KUKA KRL program: MyProgram_158().src

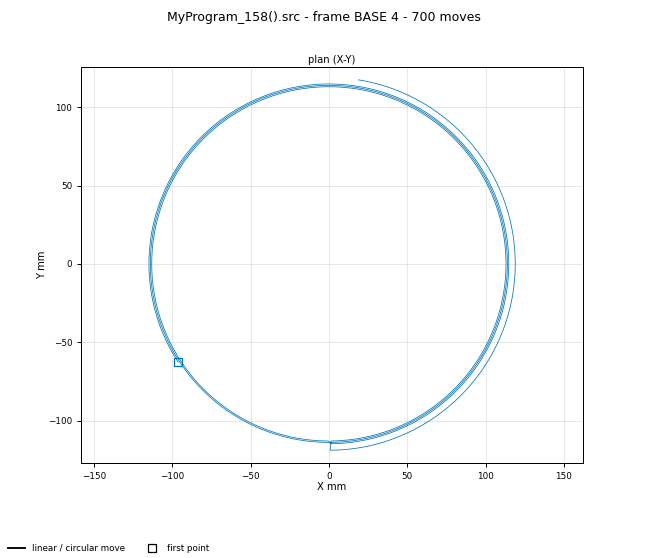
[picture p0: tool path of MyProgram_158().src in frame BASE 4, 700 of 700 moves have a stored position in this frame; points joined in program order, loops and branches not executed]
&ACCESS RVP
&REL 1
&PARAM TEMPLATE = C:\KRC\Roboter\Template\vorgabe
&PARAM EDITMASK = *
DEF MyProgram_158()
; ---- Setting reference (Base) ----
$BASE = BASE_DATA[4]

; --------------------------
; ---- Setting tool (TCP) ----
$TOOL = TOOL_DATA[3]
; --------------------------

$VEL.CP = VEL_APROX_PRINT
Startdeposition()
$VEL.CP = VEL_PRINT
LIN {X -96.1215,Y -62.8058,Z 121,A -151.3132,B 24.9534,C -1.5764,E1 24.8649,E2 237.3764} C_DIS
LIN {X -98.7062,Y -58.6591,Z 121,A -153.4833,B 24.9524,C -1.5937,E1 24.8618,E2 239.5163} C_DIS
LIN {X -100.613,Y -55.328,Z 121,A -155.5079,B 24.9524,C -1.5945,E1 24.859,E2 241.5496} C_DIS
LIN {X -102.3262,Y -52.0874,Z 121,A -157.2957,B 24.952,C -1.6013,E1 24.8567,E2 243.3308} C_DIS
LIN {X -104.3543,Y -47.8986,Z 121,A -160.2123,B 24.953,C -1.5842,E1 24.8532,E2 246.3041} C_DIS
LIN {X -106.1362,Y -43.808,Z 121,A -161.886,B 24.9513,C -1.6127,E1 24.8515,E2 247.9191} C_DIS
LIN {X -107.2271,Y -41.0641,Z 121,A -163.2123,B 24.9506,C -1.6229,E1 24.8501,E2 249.2284} C_DIS
LIN {X -108.5471,Y -37.4383,Z 121,A -165.2668,B 24.9506,C -1.6235,E1 24.8482,E2 251.2933} C_DIS
LIN {X -109.6661,Y -34.0158,Z 121,A -167.0294,B 24.9502,C -1.6304,E1 24.8467,E2 253.0496} C_DIS
LIN {X -110.6984,Y -30.4946,Z 121,A -168.9363,B 24.95,C -1.6329,E1 24.8452,E2 254.9614} C_DIS
LIN {X -111.5787,Y -27.0914,Z 121,A -170.6546,B 24.9496,C -1.6398,E1 24.8441,E2 256.6733} C_DIS
LIN {X -112.4202,Y -23.3559,Z 121,A -172.6551,B 24.9495,C -1.6422,E1 24.8429,E2 258.6799} C_DIS
LIN {X -113.0351,Y -20.1694,Z 121,A -174.8026,B 24.9504,C -1.6265,E1 24.8418,E2 260.8777} C_DIS
LIN {X -113.7096,Y -15.9343,Z 121,A -176.449,B 24.9488,C -1.6528,E1 24.8412,E2 262.4712} C_DIS
LIN {X -114.0425,Y -13.3431,Z 121,A -178.2058,B 24.9497,C -1.6391,E1 24.8406,E2 264.2712} C_DIS
LIN {X -114.4392,Y -9.3513,Z 121,A 179.6628,B 24.9496,C -1.6404,E1 24.8401,E2 266.4122} C_DIS
LIN {X -114.7175,Y -4.8606,Z 121,A 178.0279,B 24.9476,C -1.6717,E1 24.8399,E2 267.9823} C_DIS
LIN {X -114.814,Y -1.3829,Z 121,A 175.4927,B 24.9492,C -1.6459,E1 24.8399,E2 270.5943} C_DIS
LIN {X -114.7594,Y 3.7508,Z 121,A 173.0506,B 24.9484,C -1.659,E1 24.84,E2 273.02} C_DIS
LIN {X -114.514,Y 8.3994,Z 121,A 171.3096,B 24.9465,C -1.6894,E1 24.8403,E2 274.699} C_DIS
LIN {X -113.8679,Y 14.7586,Z 121,A 168.0814,B 24.946,C -1.6982,E1 24.8413,E2 277.9254} C_DIS
LIN {X -113.3453,Y 18.3552,Z 121,A 166.2551,B 24.9456,C -1.7036,E1 24.8421,E2 279.7497} C_DIS
LIN {X -112.7131,Y 21.898,Z 121,A 164.4701,B 24.9452,C -1.7098,E1 24.843,E2 281.5304} C_DIS
LIN {X -112.1059,Y 24.8216,Z 121,A 162.4049,B 24.9463,C -1.692,E1 24.8443,E2 283.6503} C_DIS
LIN {X -111.0532,Y 29.1768,Z 121,A 160.7315,B 24.9445,C -1.7213,E1 24.8454,E2 285.2636} C_DIS
LIN {X -110.14,Y 32.4493,Z 121,A 159.1356,B 24.9439,C -1.7306,E1 24.8466,E2 286.8465} C_DIS
LIN {X -107.4375,Y 40.5085,Z 121,A 154.9999,B 24.9427,C -1.7481,E1 24.8503,E2 290.964} C_DIS
LIN {X -105.096,Y 46.2461,Z 121,A 151.596,B 24.9429,C -1.7452,E1 24.854,E2 294.3938} C_DIS
LIN {X -102.9973,Y 50.7479,Z 121,A 149.1343,B 24.9424,C -1.7534,E1 24.8569,E2 296.8493} C_DIS
LIN {X -101.2249,Y 54.1999,Z 121,A 147.1466,B 24.9421,C -1.7571,E1 24.8595,E2 298.8389} C_DIS
LIN {X -96.7746,Y 61.7938,Z 121,A 142.7854,B 24.9412,C -1.771,E1 24.8658,E2 303.1894} C_DIS
LIN {X -94.9438,Y 64.5713,Z 121,A 140.5435,B 24.9424,C -1.7526,E1 24.8694,E2 305.4863} C_DIS
LIN {X -92.4138,Y 68.1437,Z 121,A 138.3387,B 24.9421,C -1.7578,E1 24.873,E2 307.6894} C_DIS
LIN {X -89.7147,Y 71.6613,Z 121,A 136.6412,B 24.9403,C -1.7841,E1 24.8758,E2 309.3321} C_DIS
LIN {X -87.3156,Y 74.5636,Z 121,A 134.8321,B 24.9398,C -1.7919,E1 24.8791,E2 311.1311} C_DIS
LIN {X -84.7529,Y 77.4644,Z 121,A 132.9066,B 24.9395,C -1.797,E1 24.8826,E2 313.0529} C_DIS
LIN {X -82.5435,Y 79.8143,Z 121,A 131.2955,B 24.9392,C -1.801,E1 24.8857,E2 314.6615} C_DIS
LIN {X -79.9211,Y 82.4406,Z 121,A 129.4166,B 24.939,C -1.8044,E1 24.8895,E2 316.5402} C_DIS
LIN {X -77.5694,Y 84.6565,Z 121,A 127.7878,B 24.9388,C -1.8075,E1 24.8928,E2 318.1682} C_DIS
LIN {X -74.6448,Y 87.2464,Z 121,A 125.8351,B 24.9385,C -1.8119,E1 24.8969,E2 320.1183} C_DIS
LIN {X -72.0721,Y 89.3835,Z 121,A 124.0608,B 24.9385,C -1.8113,E1 24.9008,E2 321.9006} C_DIS
LIN {X -68.9305,Y 91.8277,Z 121,A 122.1405,B 24.938,C -1.8182,E1 24.905,E2 323.8114} C_DIS
LIN {X -64.5217,Y 94.9774,Z 121,A 119.0522,B 24.9387,C -1.8081,E1 24.9122,E2 326.9343} C_DIS
LIN {X -61.6039,Y 96.8965,Z 121,A 117.6079,B 24.9377,C -1.8235,E1 24.9155,E2 328.3465} C_DIS
LIN {X -58.7884,Y 98.6297,Z 121,A 115.9289,B 24.9375,C -1.8254,E1 24.9195,E2 330.0263} C_DIS
LIN {X -55.2102,Y 100.6769,Z 121,A 114.0202,B 24.9369,C -1.8351,E1 24.9241,E2 331.9175} C_DIS
LIN {X -52.7307,Y 101.9975,Z 121,A 112.5738,B 24.9369,C -1.8356,E1 24.9277,E2 333.3666} C_DIS
LIN {X -50.4381,Y 103.1509,Z 121,A 110.373,B 24.9393,C -1.8001,E1 24.9335,E2 335.6574} C_DIS
LIN {X -45.2421,Y 105.5337,Z 121,A 108.4902,B 24.9363,C -1.844,E1 24.938,E2 337.4405} C_DIS
LIN {X -39.388,Y 107.8532,Z 121,A 105.2389,B 24.9363,C -1.8437,E1 24.9465,E2 340.6993} C_DIS
LIN {X -35.8676,Y 109.0758,Z 121,A 103.4013,B 24.9361,C -1.8469,E1 24.9513,E2 342.5329} C_DIS
LIN {X -32.6704,Y 110.0744,Z 121,A 101.7237,B 24.9359,C -1.8486,E1 24.9558,E2 344.2094} C_DIS
LIN {X -28.9554,Y 111.1101,Z 121,A 99.5825,B 24.9364,C -1.8415,E1 24.9616,E2 346.3706} C_DIS
LIN {X -23.8184,Y 112.3248,Z 121,A 96.5727,B 24.9373,C -1.8283,E1 24.9699,E2 349.4157} C_DIS
LIN {X -19.6037,Y 113.1365,Z 121,A 94.9134,B 24.9358,C -1.85,E1 24.9744,E2 351.025} C_DIS
LIN {X -13.3544,Y 114.0412,Z 121,A 92.0278,B 24.9349,C -1.8632,E1 24.9823,E2 353.8815} C_DIS
LIN {X -7.8614,Y 114.551,Z 121,A 89.1574,B 24.9352,C -1.8595,E1 24.9903,E2 356.762} C_DIS
LIN {X -4.8853,Y 114.7164,Z 121,A 86.9827,B 24.9372,C -1.831,E1 24.9966,E2 359.0049} C_DIS
LIN {X -0.3746,Y 114.8203,Z 121,A 85.6519,B 24.9344,C -1.8706,E1 25,E2 360.242} C_DIS
LIN {X 5.1557,Y 114.7048,Z 121,A 82.5408,B 24.9354,C -1.8558,E1 25.0088,E2 363.3874} C_DIS
LIN {X 7.8335,Y 114.5529,Z 121,A 80.6882,B 24.937,C -1.8339,E1 25.0141,E2 365.2913} C_DIS
LIN {X 12.0548,Y 114.1859,Z 121,A 78.4447,B 24.9374,C -1.8281,E1 25.0203,E2 367.5469} C_DIS
LIN {X 16.9074,Y 113.5706,Z 121,A 76.5126,B 24.9359,C -1.8491,E1 25.0255,E2 369.4275} C_DIS
LIN {X 21.8894,Y 112.7147,Z 121,A 74.2506,B 24.9352,C -1.8594,E1 25.0317,E2 371.6625} C_DIS
LIN {X 26.0769,Y 111.8203,Z 121,A 72.0876,B 24.9353,C -1.8572,E1 25.0376,E2 373.8279} C_DIS
LIN {X 29.1301,Y 111.0652,Z 121,A 70.5499,B 24.9353,C -1.8576,E1 25.0417,E2 375.3623} C_DIS
LIN {X 33.9752,Y 109.6787,Z 121,A 67.9832,B 24.9356,C -1.8535,E1 25.0486,E2 377.9344} C_DIS
LIN {X 37.6505,Y 108.4726,Z 121,A 65.9823,B 24.9359,C -1.8488,E1 25.0539,E2 379.9426} C_DIS
LIN {X 41.1905,Y 107.1792,Z 121,A 64.0737,B 24.9361,C -1.8457,E1 25.0589,E2 381.8543} C_DIS
LIN {X 44.6995,Y 105.7625,Z 121,A 62.3212,B 24.9359,C -1.8497,E1 25.0634,E2 383.5933} C_DIS
LIN {X 48.0774,Y 104.2711,Z 121,A 60.4926,B 24.9359,C -1.8482,E1 25.0681,E2 385.421} C_DIS
LIN {X 51.8809,Y 102.4318,Z 121,A 58.3052,B 24.9364,C -1.842,E1 25.0736,E2 387.6171} C_DIS
LIN {X 55.0868,Y 100.7438,Z 121,A 56.5389,B 24.9364,C -1.8414,E1 25.0779,E2 389.3798} C_DIS
LIN {X 58.2725,Y 98.9347,Z 121,A 54.7042,B 24.9366,C -1.8385,E1 25.0824,E2 391.2159} C_DIS
LIN {X 61.4356,Y 97.0046,Z 121,A 52.8073,B 24.937,C -1.8335,E1 25.0869,E2 393.1187} C_DIS
LIN {X 63.9947,Y 95.3342,Z 121,A 51.3249,B 24.937,C -1.8329,E1 25.0903,E2 394.5976} C_DIS
LIN {X 66.3478,Y 93.7116,Z 121,A 49.8719,B 24.9373,C -1.8293,E1 25.0936,E2 396.0541} C_DIS
LIN {X 69.4672,Y 91.4244,Z 121,A 46.9689,B 24.9404,C -1.7825,E1 25.1003,E2 399.0569} C_DIS
LIN {X 74.3586,Y 87.4903,Z 121,A 45.2175,B 24.9367,C -1.8382,E1 25.1038,E2 400.6701} C_DIS
LIN {X 78.1942,Y 84.0821,Z 121,A 42.2735,B 24.9382,C -1.8156,E1 25.11,E2 403.6558} C_DIS
LIN {X 80.7429,Y 81.6353,Z 121,A 40.602,B 24.9382,C -1.816,E1 25.1133,E2 405.3193} C_DIS
LIN {X 82.4406,Y 79.9211,Z 121,A 38.63,B 24.9407,C -1.7787,E1 25.1173,E2 407.3707} C_DIS
LIN {X 85.9184,Y 76.1709,Z 121,A 36.8868,B 24.9386,C -1.8094,E1 25.1204,E2 409.0339} C_DIS
LIN {X 89.5047,Y 71.9227,Z 121,A 33.9906,B 24.9395,C -1.7972,E1 25.1256,E2 411.9455} C_DIS
LIN {X 91.5655,Y 69.2794,Z 121,A 32.4088,B 24.9395,C -1.7972,E1 25.1283,E2 413.5196} C_DIS
LIN {X 93.5687,Y 66.5482,Z 121,A 30.7815,B 24.9395,C -1.7959,E1 25.1309,E2 415.1423} C_DIS
LIN {X 96.4611,Y 62.2823,Z 121,A 28.1901,B 24.9401,C -1.7883,E1 25.135,E2 417.7387} C_DIS
LIN {X 98.3019,Y 59.3344,Z 121,A 26.397,B 24.9405,C -1.781,E1 25.1376,E2 419.54} C_DIS
LIN {X 99.997,Y 56.4322,Z 121,A 24.8055,B 24.9405,C -1.7803,E1 25.1398,E2 421.1248} C_DIS
LIN {X 101.6157,Y 53.46,Z 121,A 22.5104,B 24.9427,C -1.7479,E1 25.1429,E2 423.4843} C_DIS
LIN {X 103.598,Y 49.51,Z 121,A 20.5831,B 24.9423,C -1.7543,E1 25.1452,E2 425.3861} C_DIS
LIN {X 104.9951,Y 46.4775,Z 121,A 19.1792,B 24.9418,C -1.7615,E1 25.1467,E2 426.7654} C_DIS
LIN {X 106.3722,Y 43.2284,Z 121,A 17.5035,B 24.9419,C -1.7603,E1 25.1485,E2 428.4347} C_DIS
LIN {X 107.8329,Y 39.4436,Z 121,A 15.5282,B 24.9422,C -1.7566,E1 25.1505,E2 430.4078} C_DIS
LIN {X 109.0136,Y 36.0582,Z 121,A 13.8068,B 24.9423,C -1.7543,E1 25.152,E2 432.1249} C_DIS
LIN {X 110.5926,Y 30.8741,Z 121,A 10.9602,B 24.9433,C -1.7394,E1 25.1543,E2 434.9904} C_DIS
LIN {X 111.6671,Y 26.7289,Z 121,A 8.5014,B 24.9447,C -1.7178,E1 25.156,E2 437.4858} C_DIS
LIN {X 112.4325,Y 23.296,Z 121,A 7.1876,B 24.9437,C -1.7328,E1 25.1567,E2 438.7567} C_DIS
LIN {X 112.9625,Y 20.5735,Z 121,A 5.3858,B 24.9453,C -1.709,E1 25.1576,E2 440.604} C_DIS
LIN {X 113.558,Y 16.9887,Z 121,A 3.9219,B 24.9446,C -1.7194,E1 25.1582,E2 442.0348} C_DIS
LIN {X 114.0229,Y 13.5104,Z 121,A 2.2875,B 24.9446,C -1.7193,E1 25.1588,E2 443.66} C_DIS
LIN {X 114.3753,Y 10.1102,Z 121,A 0.5482,B 24.9451,C -1.7122,E1 25.1593,E2 445.4056} C_DIS
LIN {X 114.6333,Y 6.5551,Z 121,A -1.1978,B 24.9453,C -1.708,E1 25.1596,E2 447.1512} C_DIS
LIN {X 114.7743,Y 3.2623,Z 121,A -2.8664,B 24.9457,C -1.7015,E1 25.1598,E2 448.8251} C_DIS
LIN {X 114.8185,Y -0.7449,Z 121,A -4.8494,B 24.9461,C -1.6957,E1 25.1598,E2 450.8098} C_DIS
LIN {X 114.7256,Y -4.6719,Z 121,A -6.7449,B 24.9463,C -1.6924,E1 25.1596,E2 452.702} C_DIS
LIN {X 114.5495,Y -7.8841,Z 121,A -8.3454,B 24.9466,C -1.6874,E1 25.1593,E2 454.3049} C_DIS
LIN {X 114.2214,Y -11.7158,Z 121,A -9.9878,B 24.9462,C -1.6941,E1 25.1589,E2 455.9217} C_DIS
LIN {X 113.6208,Y -16.5537,Z 121,A -13.0095,B 24.9485,C -1.6586,E1 25.1578,E2 459.0092} C_DIS
LIN {X 113.104,Y -19.7867,Z 121,A -14.3439,B 24.9479,C -1.6672,E1 25.1572,E2 460.3155} C_DIS
LIN {X 112.5322,Y -22.8105,Z 121,A -15.8061,B 24.948,C -1.6657,E1 25.1564,E2 461.7727} C_DIS
LIN {X 112.0044,Y -25.28,Z 121,A -17.0567,B 24.9482,C -1.662,E1 25.1556,E2 463.0247} C_DIS
LIN {X 111.2159,Y -28.5439,Z 121,A -18.737,B 24.9486,C -1.6564,E1 25.1545,E2 464.7084} C_DIS
LIN {X 110.2966,Y -31.9185,Z 121,A -20.5716,B 24.9492,C -1.6466,E1 25.1531,E2 466.5557} C_DIS
LIN {X 109.2307,Y -35.3889,Z 121,A -22.6194,B 24.9502,C -1.6299,E1 25.1514,E2 468.6313} C_DIS
LIN {X 108.1578,Y -38.5478,Z 121,A -24.0023,B 24.9497,C -1.6378,E1 25.1501,E2 469.9878} C_DIS
LIN {X 106.8943,Y -41.9206,Z 121,A -25.5185,B 24.9493,C -1.6453,E1 25.1486,E2 471.4778} C_DIS
LIN {X 105.7281,Y -44.781,Z 121,A -27.3593,B 24.9504,C -1.6265,E1 25.1466,E2 473.3527} C_DIS
LIN {X 102.7462,Y -51.2545,Z 121,A -30.8679,B 24.9509,C -1.6179,E1 25.1424,E2 476.8627} C_DIS
LIN {X 100.9603,Y -54.6877,Z 121,A -32.4978,B 24.9504,C -1.6262,E1 25.1403,E2 478.4645} C_DIS
LIN {X 97.0688,Y -61.3329,Z 121,A -36.5884,B 24.9518,C -1.6034,E1 25.1345,E2 482.5879} C_DIS
LIN {X 95.0203,Y -64.4584,Z 121,A -38.3723,B 24.9519,C -1.6019,E1 25.1317,E2 484.3666} C_DIS
LIN {X 92.7868,Y -67.6343,Z 121,A -40.2813,B 24.9522,C -1.5978,E1 25.1286,E2 486.2759} C_DIS
LIN {X 90.7135,Y -70.3913,Z 121,A -42.0985,B 24.9527,C -1.5886,E1 25.1255,E2 488.1061} C_DIS
LIN {X 88.3561,Y -73.3275,Z 121,A -43.8607,B 24.9527,C -1.589,E1 25.1224,E2 489.8592} C_DIS
LIN {X 86.0399,Y -76.0345,Z 121,A -45.7192,B 24.9532,C -1.5806,E1 25.119,E2 491.7291} C_DIS
LIN {X 83.5677,Y -78.7413,Z 121,A -47.4804,B 24.9532,C -1.5791,E1 25.1156,E2 493.4862} C_DIS
LIN {X 80.6526,Y -81.7245,Z 121,A -49.7015,B 24.954,C -1.5676,E1 25.1112,E2 495.7251} C_DIS
LIN {X 77.4731,Y -84.7448,Z 121,A -51.6968,B 24.9537,C -1.5712,E1 25.1072,E2 497.7036} C_DIS
LIN {X 74.7706,Y -87.1392,Z 121,A -53.5625,B 24.9542,C -1.5641,E1 25.1033,E2 499.5788} C_DIS
LIN {X 69.9227,Y -91.0746,Z 121,A -56.6293,B 24.9544,C -1.5594,E1 25.0966,E2 502.6451} C_DIS
LIN {X 66.8672,Y -93.341,Z 121,A -58.4819,B 24.9545,C -1.5575,E1 25.0924,E2 504.4957} C_DIS
LIN {X 64.0295,Y -95.3107,Z 121,A -60.3186,B 24.9551,C -1.5489,E1 25.0881,E2 506.3466} C_DIS
LIN {X 60.7768,Y -97.4161,Z 121,A -62.1258,B 24.9549,C -1.5509,E1 25.0839,E2 508.1433} C_DIS
LIN {X 57.5124,Y -99.379,Z 121,A -63.84,B 24.9546,C -1.5558,E1 25.0798,E2 509.8404} C_DIS
LIN {X 54.723,Y -100.9412,Z 121,A -66.578,B 24.9578,C -1.5015,E1 25.0728,E2 512.6989} C_DIS
LIN {X 49.393,Y -103.6542,Z 121,A -68.4656,B 24.9552,C -1.5458,E1 25.0683,E2 514.4767} C_DIS
LIN {X 42.3067,Y -106.7426,Z 121,A -72.4489,B 24.9559,C -1.5343,E1 25.0581,E2 518.4777} C_DIS
LIN {X 39.0113,Y -107.9906,Z 121,A -74.2842,B 24.9562,C -1.5285,E1 25.0532,E2 520.323} C_DIS
LIN {X 35.716,Y -109.1249,Z 121,A -75.866,B 24.956,C -1.5333,E1 25.0491,E2 521.8902} C_DIS
LIN {X 30.3415,Y -110.7397,Z 121,A -78.6548,B 24.9561,C -1.5307,E1 25.0416,E2 524.6806} C_DIS
LIN {X 27.6754,Y -111.4362,Z 121,A -80.0133,B 24.9561,C -1.53,E1 25.0379,E2 526.0386} C_DIS
LIN {X 21.6881,Y -112.7535,Z 121,A -83.0024,B 24.9561,C -1.5303,E1 25.0298,E2 529.023} C_DIS
LIN {X 15.8742,Y -113.7181,Z 121,A -86.1649,B 24.9568,C -1.5183,E1 25.021,E2 532.211} C_DIS
LIN {X 11.583,Y -114.2353,Z 121,A -88.3362,B 24.9569,C -1.5163,E1 25.015,E2 534.3853} C_DIS
LIN {X 7.9927,Y -114.5422,Z 121,A -89.9911,B 24.9566,C -1.5218,E1 25.0104,E2 536.0265} C_DIS
LIN {X 5.0588,Y -114.709,Z 121,A -91.4832,B 24.9567,C -1.5201,E1 25.0062,E2 537.5222} C_DIS
LIN {X 1.4985,Y -114.8123,Z 121,A -93.3515,B 24.957,C -1.5155,E1 25.001,E2 539.4009} C_DIS
LIN {X 1.4985,Y -114.8123,Z 121,A -93.3515,B 24.957,C -1.5155,E1 25.001,E2 539.4009} C_DIS
Enddeposition()
LIN {X 0.8205,Y -113.9352,Z 121,A -93.6003,B 24.9559,C -1.5349,E1 25.0004,E2 539.6037} C_DIS
Startdeposition()
$VEL.CP = VEL_PRINT
LIN {X 4.8717,Y -113.8345,Z 121,A -90.8478,B 24.954,C -1.5668,E1 25.0083,E2 536.7761} C_DIS
LIN {X 8.1536,Y -113.6476,Z 121,A -89.0673,B 24.9536,C -1.5732,E1 25.0133,E2 534.9813} C_DIS
LIN {X 14.6994,Y -112.9866,Z 121,A -86.2906,B 24.9549,C -1.5515,E1 25.0209,E2 532.2578} C_DIS
LIN {X 20.9577,Y -111.9963,Z 121,A -82.4435,B 24.953,C -1.5833,E1 25.0317,E2 528.3394} C_DIS
LIN {X 26.0634,Y -110.9185,Z 121,A -80.1548,B 24.9538,C -1.5707,E1 25.0378,E2 526.0835} C_DIS
LIN {X 29.0685,Y -110.1703,Z 121,A -78.6045,B 24.9538,C -1.572,E1 25.042,E2 524.5326} C_DIS
LIN {X 32.1861,Y -109.2984,Z 121,A -76.7232,B 24.9529,C -1.5852,E1 25.0471,E2 522.6231} C_DIS
LIN {X 36.1944,Y -108.0373,Z 121,A -74.8013,B 24.9533,C -1.5792,E1 25.0522,E2 520.719} C_DIS
LIN {X 39.2027,Y -106.9823,Z 121,A -73.2543,B 24.9533,C -1.5788,E1 25.0562,E2 519.1763} C_DIS
LIN {X 42.4649,Y -105.731,Z 121,A -70.9958,B 24.9518,C -1.604,E1 25.0623,E2 516.863} C_DIS
LIN {X 45.7854,Y -104.3351,Z 121,A -69.8746,B 24.9535,C -1.5754,E1 25.065,E2 515.8122} C_DIS
LIN {X 47.9547,Y -103.3557,Z 121,A -68.446,B 24.9528,C -1.5878,E1 25.0686,E2 514.358} C_DIS
LIN {X 51.2356,Y -101.7713,Z 121,A -66.5435,B 24.9524,C -1.594,E1 25.0734,E2 512.4459} C_DIS
LIN {X 56.7317,Y -98.8107,Z 121,A -63.5306,B 24.9524,C -1.5938,E1 25.0808,E2 509.4423} C_DIS
LIN {X 59.3692,Y -97.2491,Z 121,A -61.9362,B 24.9521,C -1.5991,E1 25.0846,E2 507.8403} C_DIS
LIN {X 62.7529,Y -95.1005,Z 121,A -59.9229,B 24.9519,C -1.6029,E1 25.0893,E2 505.8244} C_DIS
LIN {X 65.6081,Y -93.1563,Z 121,A -58.2849,B 24.9519,C -1.6019,E1 25.0931,E2 504.1945} C_DIS
LIN {X 67.4533,Y -91.8265,Z 121,A -57.1559,B 24.9519,C -1.6037,E1 25.0956,E2 503.0654} C_DIS
LIN {X 70.0049,Y -89.8982,Z 121,A -55.2667,B 24.9508,C -1.6201,E1 25.0999,E2 501.1442} C_DIS
LIN {X 72.7486,Y -87.6908,Z 121,A -53.7199,B 24.9512,C -1.6137,E1 25.1032,E2 499.6184} C_DIS
LIN {X 75.2244,Y -85.5772,Z 121,A -52.1275,B 24.9512,C -1.6154,E1 25.1065,E2 498.0282} C_DIS
LIN {X 77.8308,Y -83.2136,Z 121,A -50.3206,B 24.9507,C -1.6214,E1 25.1102,E2 496.2146} C_DIS
LIN {X 80.3573,Y -80.7768,Z 121,A -48.5194,B 24.9504,C -1.6274,E1 25.1139,E2 494.4068} C_DIS
LIN {X 82.9044,Y -78.1595,Z 121,A -46.7179,B 24.9502,C -1.6304,E1 25.1173,E2 492.606} C_DIS
LIN {X 85.3032,Y -75.5366,Z 121,A -44.9087,B 24.9498,C -1.636,E1 25.1207,E2 490.7917} C_DIS
LIN {X 87.6544,Y -72.7924,Z 121,A -43.1734,B 24.9498,C -1.637,E1 25.1238,E2 489.0619} C_DIS
LIN {X 90.0625,Y -69.7916,Z 121,A -41.2018,B 24.9494,C -1.6439,E1 25.1273,E2 487.0832} C_DIS
LIN {X 92.1074,Y -67.0697,Z 121,A -39.4465,B 24.9489,C -1.6507,E1 25.1302,E2 485.3205} C_DIS
LIN {X 94.3298,Y -63.9056,Z 121,A -37.6308,B 24.9489,C -1.6501,E1 25.133,E2 483.5149} C_DIS
LIN {X 96.2633,Y -60.9581,Z 121,A -35.3486,B 24.9472,C -1.6791,E1 25.1366,E2 481.1758} C_DIS
LIN {X 98.2144,Y -57.7583,Z 121,A -34.0632,B 24.9486,C -1.6565,E1 25.1383,E2 479.9504} C_DIS
LIN {X 99.7805,Y -55.0116,Z 121,A -32.3301,B 24.9479,C -1.6678,E1 25.1407,E2 478.1995} C_DIS
LIN {X 101.4819,Y -51.8022,Z 121,A -30.5741,B 24.9477,C -1.67,E1 25.1429,E2 476.4476} C_DIS
LIN {X 103.0768,Y -48.5539,Z 121,A -28.7404,B 24.9473,C -1.6762,E1 25.1452,E2 474.6093} C_DIS
LIN {X 104.1791,Y -46.1408,Z 121,A -26.8822,B 24.9455,C -1.705,E1 25.1473,E2 472.6932} C_DIS
LIN {X 105.809,Y -42.2721,Z 121,A -25.4248,B 24.9471,C -1.6807,E1 25.1488,E2 471.3011} C_DIS
LIN {X 107.3612,Y -38.155,Z 121,A -23.0019,B 24.946,C -1.6975,E1 25.1512,E2 468.8521} C_DIS
LIN {X 108.5245,Y -34.7077,Z 121,A -21.296,B 24.946,C -1.6975,E1 25.1526,E2 467.156} C_DIS
LIN {X 109.6168,Y -31.0834,Z 121,A -19.4564,B 24.9458,C -1.7006,E1 25.1541,E2 465.3196} C_DIS
LIN {X 110.5867,Y -27.4373,Z 121,A -17.4915,B 24.9452,C -1.7099,E1 25.1554,E2 463.3442} C_DIS
LIN {X 111.4834,Y -23.5347,Z 121,A -15.2824,B 24.9442,C -1.7256,E1 25.1568,E2 461.1109} C_DIS
LIN {X 112.7984,Y -16.0799,Z 121,A -11.1815,B 24.9425,C -1.7519,E1 25.1586,E2 456.972} C_DIS
LIN {X 113.3242,Y -11.8177,Z 121,A -10.0291,B 24.9451,C -1.7115,E1 25.159,E2 455.9218} C_DIS
LIN {X 113.5561,Y -9.3336,Z 121,A -8.3643,B 24.9436,C -1.7348,E1 25.1594,E2 454.2119} C_DIS
LIN {X 113.7921,Y -5.7983,Z 121,A -6.5206,B 24.943,C -1.7435,E1 25.1596,E2 452.3586} C_DIS
LIN {X 113.9196,Y -2.0886,Z 121,A -4.7521,B 24.943,C -1.745,E1 25.1598,E2 450.5971} C_DIS
LIN {X 113.9348,Y 1.0341,Z 121,A -3.2861,B 24.943,C -1.7452,E1 25.1598,E2 449.1393} C_DIS
LIN {X 113.878,Y 3.7263,Z 121,A -1.8071,B 24.9422,C -1.7555,E1 25.1596,E2 447.6448} C_DIS
LIN {X 113.6851,Y 7.5992,Z 121,A 0.0875,B 24.942,C -1.7592,E1 25.1593,E2 445.7528} C_DIS
LIN {X 113.4035,Y 11.0462,Z 121,A 1.9165,B 24.9413,C -1.769,E1 25.1589,E2 443.9114} C_DIS
LIN {X 113.0167,Y 14.4666,Z 121,A 3.5248,B 24.9413,C -1.7688,E1 25.1583,E2 442.3131} C_DIS
LIN {X 112.2124,Y 19.7633,Z 121,A 6.0098,B 24.9414,C -1.7676,E1 25.1573,E2 439.8456} C_DIS
LIN {X 111.6915,Y 22.5212,Z 121,A 7.9849,B 24.9394,C -1.7985,E1 25.1562,E2 437.8092} C_DIS
LIN {X 110.9895,Y 25.756,Z 121,A 9.2831,B 24.9402,C -1.7865,E1 25.1554,E2 436.5468} C_DIS
LIN {X 110.1215,Y 29.2494,Z 121,A 11.0748,B 24.9399,C -1.7912,E1 25.1541,E2 434.7543} C_DIS
LIN {X 109.2142,Y 32.47,Z 121,A 12.935,B 24.939,C -1.8047,E1 25.1526,E2 432.8729} C_DIS
LIN {X 107.9595,Y 36.425,Z 121,A 14.8383,B 24.9391,C -1.8025,E1 25.151,E2 430.9856} C_DIS
LIN {X 106.8849,Y 39.4696,Z 121,A 16.5033,B 24.9386,C -1.8092,E1 25.1494,E2 429.314} C_DIS
LIN {X 105.5697,Y 42.8612,Z 121,A 18.2233,B 24.9386,C -1.8096,E1 25.1476,E2 427.6028} C_DIS
LIN {X 104.2454,Y 45.9911,Z 121,A 20.0191,B 24.938,C -1.8186,E1 25.1456,E2 425.7956} C_DIS
LIN {X 102.88,Y 48.9685,Z 121,A 21.6142,B 24.9379,C -1.8208,E1 25.1438,E2 424.2037} C_DIS
LIN {X 100.9849,Y 52.7657,Z 121,A 23.5188,B 24.9382,C -1.8162,E1 25.1414,E2 422.3201} C_DIS
LIN {X 99.9054,Y 54.7834,Z 121,A 24.7524,B 24.9377,C -1.8232,E1 25.1397,E2 421.0765} C_DIS
LIN {X 98.3602,Y 57.5117,Z 121,A 26.4304,B 24.9371,C -1.8322,E1 25.1374,E2 419.386} C_DIS
LIN {X 96.6157,Y 60.394,Z 121,A 28.0751,B 24.9369,C -1.8344,E1 25.135,E2 417.7443} C_DIS
LIN {X 94.6297,Y 63.4626,Z 121,A 29.9975,B 24.9363,C -1.8431,E1 25.132,E2 415.811} C_DIS
LIN {X 92.5968,Y 66.3923,Z 121,A 31.7305,B 24.9362,C -1.8449,E1 25.1292,E2 414.0823} C_DIS
LIN {X 90.7716,Y 68.8683,Z 121,A 33.1408,B 24.9364,C -1.8425,E1 25.1269,E2 412.6845} C_DIS
LIN {X 89.0614,Y 71.0661,Z 121,A 34.6094,B 24.9359,C -1.849,E1 25.1243,E2 411.2074} C_DIS
LIN {X 86.463,Y 74.2048,Z 121,A 36.5771,B 24.9359,C -1.8501,E1 25.1208,E2 409.246} C_DIS
LIN {X 84.405,Y 76.5394,Z 121,A 38.7713,B 24.9336,C -1.8825,E1 25.1166,E2 406.9849} C_DIS
LIN {X 81.6222,Y 79.4997,Z 121,A 40.1681,B 24.9353,C -1.8574,E1 25.114,E2 405.6535} C_DIS
LIN {X 79.7879,Y 81.3393,Z 121,A 41.5629,B 24.9348,C -1.8643,E1 25.1112,E2 404.2484} C_DIS
LIN {X 77.1288,Y 83.8642,Z 121,A 43.6492,B 24.9338,C -1.8791,E1 25.1069,E2 402.1355} C_DIS
LIN {X 73.648,Y 86.9374,Z 121,A 45.8283,B 24.934,C -1.8767,E1 25.1023,E2 399.9708} C_DIS
LIN {X 69.2364,Y 90.4904,Z 121,A 48.4979,B 24.9342,C -1.8738,E1 25.0965,E2 397.3178} C_DIS
LIN {X 66.9351,Y 92.2059,Z 121,A 50.0829,B 24.9335,C -1.8828,E1 25.0929,E2 395.7174} C_DIS
LIN {X 63.4306,Y 94.6514,Z 121,A 52.1981,B 24.9335,C -1.8848,E1 25.088,E2 393.6044} C_DIS
LIN {X 60.4394,Y 96.5874,Z 121,A 53.919,B 24.9335,C -1.8845,E1 25.084,E2 391.8899} C_DIS
LIN {X 57.3985,Y 98.4271,Z 121,A 55.8519,B 24.9328,C -1.8937,E1 25.0793,E2 389.9412} C_DIS
LIN {X 54.0357,Y 100.3109,Z 121,A 57.5374,B 24.9334,C -1.8851,E1 25.0752,E2 388.2809} C_DIS
LIN {X 51.6657,Y 101.5516,Z 121,A 59.0741,B 24.9327,C -1.8954,E1 25.0714,E2 386.724} C_DIS
LIN {X 48.0244,Y 103.3232,Z 121,A 61.0163,B 24.9327,C -1.8937,E1 25.0665,E2 384.7909} C_DIS
LIN {X 45.0519,Y 104.6548,Z 121,A 62.6773,B 24.9326,C -1.8965,E1 25.0622,E2 383.1273} C_DIS
LIN {X 41.5876,Y 106.0778,Z 121,A 64.5464,B 24.9325,C -1.8979,E1 25.0574,E2 381.2593} C_DIS
LIN {X 38.4499,Y 107.2568,Z 121,A 66.3212,B 24.9321,C -1.9033,E1 25.0527,E2 379.4752} C_DIS
LIN {X 34.9809,Y 108.436,Z 121,A 68.1082,B 24.9321,C -1.9025,E1 25.048,E2 377.6937} C_DIS
LIN {X 30.855,Y 109.6816,Z 121,A 70.2293,B 24.9321,C -1.902,E1 25.0423,E2 375.5772} C_DIS
LIN {X 27.0779,Y 110.6744,Z 121,A 72.246,B 24.9319,C -1.9055,E1 25.0368,E2 373.5553} C_DIS
LIN {X 22.7495,Y 111.6446,Z 121,A 74.4083,B 24.9321,C -1.9036,E1 25.031,E2 371.4003} C_DIS
LIN {X 19.7316,Y 112.218,Z 121,A 76.1671,B 24.9314,C -1.9135,E1 25.0261,E2 369.6199} C_DIS
LIN {X 15.0523,Y 112.9408,Z 121,A 78.7134,B 24.9308,C -1.9214,E1 25.019,E2 367.0573} C_DIS
LIN {X 11.7201,Y 113.3344,Z 121,A 79.5587,B 24.9334,C -1.8852,E1 25.0169,E2 366.2982} C_DIS
LIN {X 5.662,Y 113.7997,Z 121,A 84.0849,B 24.9288,C -1.9489,E1 25.0039,E2 361.623} C_DIS
LIN {X -0.4418,Y 113.9382,Z 121,A 85.8691,B 24.9328,C -1.8928,E1 24.9992,E2 359.972} C_DIS
LIN {X -6.1547,Y 113.7724,Z 121,A 88.9515,B 24.9323,C -1.9008,E1 24.9906,E2 356.8702} C_DIS
LIN {X -12.9858,Y 113.1966,Z 121,A 92.2052,B 24.933,C -1.8908,E1 24.9816,E2 353.6385} C_DIS
LIN {X -16.5485,Y 112.7318,Z 121,A 94.2887,B 24.9322,C -1.9013,E1 24.9757,E2 351.5284} C_DIS
LIN {X -20.2226,Y 112.1297,Z 121,A 96.1516,B 24.9324,C -1.8996,E1 24.9706,E2 349.6679} C_DIS
LIN {X -23.6736,Y 111.4539,Z 121,A 98.4216,B 24.9309,C -1.9193,E1 24.9643,E2 347.3484} C_DIS
LIN {X -27.3944,Y 110.5972,Z 121,A 99.7997,B 24.9327,C -1.8946,E1 24.9607,E2 346.0271} C_DIS
LIN {X -30.939,Y 109.6578,Z 121,A 101.6347,B 24.9329,C -1.8923,E1 24.9558,E2 344.1947} C_DIS
LIN {X -34.2088,Y 108.6831,Z 121,A 103.3469,B 24.933,C -1.8902,E1 24.9512,E2 342.4846} C_DIS
LIN {X -36.6489,Y 107.884,Z 121,A 104.7836,B 24.9327,C -1.8947,E1 24.9474,E2 341.0345} C_DIS
LIN {X -41.8093,Y 105.9907,Z 121,A 107.3057,B 24.9337,C -1.8809,E1 24.9408,E2 338.5399} C_DIS
LIN {X -44.1872,Y 105.0216,Z 121,A 108.7617,B 24.9333,C -1.8859,E1 24.937,E2 337.0686} C_DIS
LIN {X -47.3009,Y 103.6578,Z 121,A 110.7964,B 24.9326,C -1.8968,E1 24.9318,E2 335.0031} C_DIS
LIN {X -51.809,Y 101.4784,Z 121,A 112.9392,B 24.9339,C -1.8772,E1 24.9265,E2 332.9012} C_DIS
LIN {X -54.6624,Y 99.971,Z 121,A 114.5705,B 24.9341,C -1.8748,E1 24.9225,E2 331.2713} C_DIS
LIN {X -57.5174,Y 98.3568,Z 121,A 116.7333,B 24.9328,C -1.893,E1 24.9172,E2 329.0586} C_DIS
LIN {X -60.5092,Y 96.5437,Z 121,A 118.0957,B 24.9342,C -1.8733,E1 24.914,E2 327.7387} C_DIS
LIN {X -65.9343,Y 92.9236,Z 121,A 121.9125,B 24.9331,C -1.8888,E1 24.9051,E2 323.872} C_DIS
LIN {X -69.2376,Y 90.4895,Z 121,A 123.2273,B 24.9356,C -1.8538,E1 24.9024,E2 322.6361} C_DIS
LIN {X -72.2869,Y 88.0745,Z 121,A 125.4946,B 24.935,C -1.8621,E1 24.8974,E2 320.3404} C_DIS
LIN {X -74.9878,Y 85.7839,Z 121,A 127.1684,B 24.9356,C -1.8538,E1 24.8939,E2 318.6799} C_DIS
LIN {X -77.5093,Y 83.515,Z 121,A 129.029,B 24.9354,C -1.856,E1 24.89,E2 316.8065} C_DIS
LIN {X -80.1577,Y 80.974,Z 121,A 130.7536,B 24.9361,C -1.8467,E1 24.8866,E2 315.0969} C_DIS
LIN {X -82.6908,Y 78.3867,Z 121,A 132.639,B 24.9362,C -1.8448,E1 24.8829,E2 313.2079} C_DIS
LIN {X -85.0666,Y 75.8009,Z 121,A 134.4144,B 24.9365,C -1.8407,E1 24.8796,E2 311.4343} C_DIS
LIN {X -87.5827,Y 72.8787,Z 121,A 136.2843,B 24.937,C -1.8328,E1 24.8763,E2 309.5746} C_DIS
LIN {X -91.698,Y 67.6289,Z 121,A 139.5059,B 24.938,C -1.8184,E1 24.8708,E2 306.3721} C_DIS
LIN {X -93.5109,Y 65.0979,Z 121,A 141.2462,B 24.9378,C -1.8211,E1 24.868,E2 304.6169} C_DIS
LIN {X -95.3465,Y 62.3798,Z 121,A 142.9576,B 24.938,C -1.8189,E1 24.8653,E2 302.9021} C_DIS
LIN {X -97.209,Y 59.435,Z 121,A 145.1164,B 24.9372,C -1.8303,E1 24.8621,E2 300.7052} C_DIS
LIN {X -99.0349,Y 56.3414,Z 121,A 146.3846,B 24.939,C -1.8033,E1 24.8604,E2 299.4946} C_DIS
LIN {X -100.4684,Y 53.7454,Z 121,A 148.0849,B 24.9388,C -1.8073,E1 24.8581,E2 297.7759} C_DIS
LIN {X -102.1232,Y 50.5261,Z 121,A 149.832,B 24.9393,C -1.7989,E1 24.8559,E2 296.0393} C_DIS
LIN {X -103.5557,Y 47.5251,Z 121,A 151.4427,B 24.9399,C -1.7914,E1 24.854,E2 294.4379} C_DIS
LIN {X -104.5039,Y 45.3981,Z 121,A 153,B 24.939,C -1.8033,E1 24.8523,E2 292.8436} C_DIS
LIN {X -106.3204,Y 40.9688,Z 121,A 155.1968,B 24.9401,C -1.7874,E1 24.85,E2 290.6724} C_DIS
LIN {X -107.5278,Y 37.6804,Z 121,A 157.5576,B 24.9389,C -1.8059,E1 24.8478,E2 288.254} C_DIS
LIN {X -108.9622,Y 33.3087,Z 121,A 159.0936,B 24.9415,C -1.7674,E1 24.8466,E2 286.801} C_DIS
LIN {X -109.6747,Y 30.8792,Z 121,A 160.4812,B 24.9415,C -1.7679,E1 24.8455,E2 285.4041} C_DIS
LIN {X -110.4041,Y 28.1602,Z 121,A 162.009,B 24.9415,C -1.7679,E1 24.8444,E2 283.8675} C_DIS
LIN {X -111.082,Y 25.3555,Z 121,A 163.4904,B 24.9417,C -1.7644,E1 24.8435,E2 282.3858} C_DIS
LIN {X -111.8503,Y 21.7159,Z 121,A 165.2697,B 24.9423,C -1.7547,E1 24.8425,E2 280.619} C_DIS
LIN {X -112.3761,Y 18.8057,Z 121,A 166.7931,B 24.9425,C -1.7514,E1 24.8418,E2 279.0946} C_DIS
LIN {X -112.8541,Y 15.6877,Z 121,A 168.4646,B 24.9426,C -1.7496,E1 24.8411,E2 277.4173} C_DIS
LIN {X -113.3732,Y 11.3493,Z 121,A 170.4729,B 24.9436,C -1.7349,E1 24.8405,E2 275.432} C_DIS
LIN {X -113.5992,Y 8.7941,Z 121,A 171.8258,B 24.9437,C -1.7332,E1 24.8402,E2 274.075} C_DIS
LIN {X -113.871,Y 3.9548,Z 121,A 174.1661,B 24.9445,C -1.7214,E1 24.8399,E2 271.7489} C_DIS
LIN {X -113.9375,Y 0.6429,Z 121,A 175.9966,B 24.9444,C -1.7225,E1 24.8398,E2 269.9047} C_DIS
LIN {X -113.9066,Y -2.7947,Z 121,A 177.8224,B 24.9445,C -1.7208,E1 24.8398,E2 268.072} C_DIS
LIN {X -113.7683,Y -6.2304,Z 121,A 179.4747,B 24.9451,C -1.7121,E1 24.8401,E2 266.4304} C_DIS
LIN {X -113.4655,Y -10.374,Z 121,A -178.3464,B 24.9453,C -1.709,E1 24.8406,E2 264.2459} C_DIS
LIN {X -113.0842,Y -13.9453,Z 121,A -176.4659,B 24.9454,C -1.7061,E1 24.8412,E2 262.361} C_DIS
LIN {X -112.5972,Y -17.4329,Z 121,A -174.607,B 24.9456,C -1.704,E1 24.842,E2 260.4959} C_DIS
LIN {X -112.0392,Y -20.726,Z 121,A -172.9927,B 24.9461,C -1.6961,E1 24.8428,E2 258.8911} C_DIS
LIN {X -111.3053,Y -24.3549,Z 121,A -171.1811,B 24.9466,C -1.6882,E1 24.8438,E2 257.0875} C_DIS
LIN {X -110.3709,Y -28.2898,Z 121,A -169.2134,B 24.9472,C -1.6793,E1 24.8451,E2 255.1296} C_DIS
LIN {X -109.5097,Y -31.4614,Z 121,A -167.4083,B 24.9471,C -1.6803,E1 24.8465,E2 253.3116} C_DIS
LIN {X -108.2775,Y -35.4708,Z 121,A -165.4546,B 24.9479,C -1.6676,E1 24.8481,E2 251.3769} C_DIS
LIN {X -107.4427,Y -37.9229,Z 121,A -163.5411,B 24.9466,C -1.6885,E1 24.85,E2 249.4029} C_DIS
LIN {X -106.0343,Y -41.6985,Z 121,A -162.449,B 24.9493,C -1.6447,E1 24.851,E2 248.4089} C_DIS
LIN {X -103.5003,Y -47.6441,Z 121,A -158.8258,B 24.949,C -1.6502,E1 24.855,E2 244.7527} C_DIS
LIN {X -102.1356,Y -50.5012,Z 121,A -157.1568,B 24.949,C -1.6488,E1 24.857,E2 243.0779} C_DIS
LIN {X -100.6754,Y -53.3533,Z 121,A -155.6537,B 24.9496,C -1.6399,E1 24.8589,E2 241.5879} C_DIS
LIN {X -99.1636,Y -56.1149,Z 121,A -153.8516,B 24.9493,C -1.6445,E1 24.8614,E2 239.7656} C_DIS
LIN {X -97.3532,Y -59.1979,Z 121,A -150.9983,B 24.9469,C -1.6831,E1 24.8658,E2 236.8055} C_DIS
LIN {X -93.7012,Y -64.8242,Z 121,A -149.0235,B 24.951,C -1.6169,E1 24.8686,E2 234.9788} C_DIS
LIN {X -91.7129,Y -67.6086,Z 121,A -147.0262,B 24.9506,C -1.6238,E1 24.8719,E2 232.9552} C_DIS
LIN {X -89.2123,Y -70.8751,Z 121,A -144.8326,B 24.9506,C -1.6239,E1 24.8757,E2 230.7509} C_DIS
LIN {X -86.6818,Y -73.9479,Z 121,A -142.9056,B 24.9511,C -1.6161,E1 24.8791,E2 228.8337} C_DIS
LIN {X -83.9208,Y -77.0671,Z 121,A -140.9235,B 24.9516,C -1.6068,E1 24.8828,E2 226.8651} C_DIS
LIN {X -81.9515,Y -79.158,Z 121,A -139.3914,B 24.9516,C -1.6072,E1 24.8858,E2 225.3252} C_DIS
LIN {X -78.9184,Y -82.1825,Z 121,A -137.3424,B 24.9521,C -1.5983,E1 24.8898,E2 223.2888} C_DIS
LIN {X -76.8649,Y -84.1063,Z 121,A -135.7117,B 24.9518,C -1.6043,E1 24.8932,E2 221.6372} C_DIS
LIN {X -73.901,Y -86.7218,Z 121,A -133.7434,B 24.9521,C -1.5996,E1 24.8974,E2 219.6724} C_DIS
LIN {X -70.6643,Y -89.3789,Z 121,A -131.7243,B 24.9525,C -1.5921,E1 24.9017,E2 217.6636} C_DIS
LIN {X -67.9975,Y -91.4258,Z 121,A -129.8533,B 24.9522,C -1.5966,E1 24.9059,E2 215.7753} C_DIS
LIN {X -64.9788,Y -93.5937,Z 121,A -128.1379,B 24.9528,C -1.587,E1 24.9098,E2 214.0767} C_DIS
LIN {X -62.4716,Y -95.286,Z 121,A -126.5169,B 24.9528,C -1.5887,E1 24.9136,E2 212.4463} C_DIS
LIN {X -56.3731,Y -99.0167,Z 121,A -122.8623,B 24.9528,C -1.5859,E1 24.9224,E2 208.7872} C_DIS
LIN {X -52.5507,Y -101.0981,Z 121,A -120.6666,B 24.953,C -1.5833,E1 24.9278,E2 206.5917} C_DIS
LIN {X -48.9828,Y -102.8731,Z 121,A -118.8317,B 24.9536,C -1.5737,E1 24.9323,E2 204.7748} C_DIS
LIN {X -46.1634,Y -104.1703,Z 121,A -116.878,B 24.9527,C -1.5886,E1 24.9374,E2 202.7808} C_DIS
LIN {X -42.3082,Y -105.7948,Z 121,A -115.1449,B 24.9538,C -1.5706,E1 24.9418,E2 201.0865} C_DIS
LIN {X -39.1617,Y -106.9972,Z 121,A -113.3769,B 24.9537,C -1.5723,E1 24.9464,E2 199.311} C_DIS
LIN {X -35.4467,Y -108.2853,Z 121,A -111.2519,B 24.9534,C -1.577,E1 24.9521,E2 197.1709} C_DIS
LIN {X -31.9796,Y -109.3596,Z 121,A -109.6578,B 24.9541,C -1.5657,E1 24.9563,E2 195.6008} C_DIS
LIN {X -29.7369,Y -109.9898,Z 121,A -108.3767,B 24.9538,C -1.5697,E1 24.9598,E2 194.3083} C_DIS
LIN {X -25.9538,Y -110.9438,Z 121,A -106.4818,B 24.9541,C -1.5657,E1 24.9649,E2 192.4202} C_DIS
LIN {X -22.8253,Y -111.629,Z 121,A -104.7098,B 24.9537,C -1.572,E1 24.9698,E2 190.6311} C_DIS
LIN {X -19.2398,Y -112.3035,Z 121,A -102.2635,B 24.9521,C -1.5982,E1 24.9767,E2 188.1204} C_DIS
LIN {X -14.3835,Y -113.0275,Z 121,A -100.1389,B 24.9531,C -1.5825,E1 24.9825,E2 186.0313} C_DIS
LIN {X -10.9397,Y -113.4133,Z 121,A -98.9612,B 24.9545,C -1.5576,E1 24.9856,E2 184.912} C_DIS
LIN {X -6.2993,Y -113.7644,Z 121,A -96.4166,B 24.954,C -1.5666,E1 24.9928,E2 182.3452} C_DIS
LIN {X -2.7614,Y -113.9072,Z 121,A -94.5522,B 24.9538,C -1.5705,E1 24.998,E2 180.4713} C_DIS
LIN {X 0.8205,Y -113.9352,Z 121,A -93.5978,B 24.9559,C -1.5339,E1 25.0004,E2 179.6037} C_DIS
Enddeposition()
LIN {X 0.8205,Y -113.9352,Z 121,A -93.5978,B 24.9559,C -1.5339,E1 25.0004,E2 179.6037} C_DIS
Startdeposition()
$VEL.CP = VEL_PRINT
LIN {X -0.3464,Y -113.057,Z 121,A -94.1938,B 24.955,C -1.549,E1 24.9989,E2 180.1637} C_DIS
LIN {X -3.1191,Y -113.0145,Z 121,A -95.4413,B 24.9547,C -1.5556,E1 24.9954,E2 181.3958} C_DIS
LIN {X -5.5458,Y -112.9231,Z 121,A -96.9543,B 24.9554,C -1.5434,E1 24.9911,E2 182.9382} C_DIS
LIN {X -8.5827,Y -112.7316,Z 121,A -98.4809,B 24.9554,C -1.544,E1 24.9869,E2 184.4638} C_DIS
LIN {X -11.6123,Y -112.4592,Z 121,A -99.8963,B 24.955,C -1.5496,E1 24.983,E2 185.8668} C_DIS
LIN {X -13.9379,Y -112.1962,Z 121,A -101.2076,B 24.9553,C -1.5444,E1 24.9793,E2 187.1912} C_DIS
LIN {X -16.967,Y -111.7771,Z 121,A -102.4901,B 24.9546,C -1.5561,E1 24.9758,E2 188.4469} C_DIS
LIN {X -19.6657,Y -111.3341,Z 121,A -103.8937,B 24.9546,C -1.5558,E1 24.9719,E2 189.8526} C_DIS
LIN {X -22.4058,Y -110.8151,Z 121,A -105.4501,B 24.955,C -1.5503,E1 24.9676,E2 191.4239} C_DIS
LIN {X -24.7753,Y -110.3112,Z 121,A -106.8096,B 24.9553,C -1.5453,E1 24.9639,E2 192.797} C_DIS
LIN {X -27.4806,Y -109.6685,Z 121,A -108.1658,B 24.9551,C -1.5483,E1 24.9602,E2 194.1479} C_DIS
LIN {X -30.1573,Y -108.9629,Z 121,A -109.6216,B 24.9551,C -1.5469,E1 24.9563,E2 195.6092} C_DIS
LIN {X -33.1415,Y -108.091,Z 121,A -110.9266,B 24.9544,C -1.5594,E1 24.9529,E2 196.8866} C_DIS
LIN {X -35.7965,Y -107.241,Z 121,A -112.4895,B 24.9547,C -1.5542,E1 24.9487,E2 198.4647} C_DIS
LIN {X -39.3971,Y -105.9728,Z 121,A -114.427,B 24.9547,C -1.5558,E1 24.9436,E2 200.4023} C_DIS
LIN {X -41.9808,Y -104.9761,Z 121,A -115.8348,B 24.9546,C -1.557,E1 24.9399,E2 201.8103} C_DIS
LIN {X -45.6069,Y -103.4511,Z 121,A -117.98,B 24.9548,C -1.5529,E1 24.9344,E2 203.9704} C_DIS
LIN {X -48.3495,Y -102.1992,Z 121,A -119.4885,B 24.9547,C -1.5554,E1 24.9306,E2 205.4766} C_DIS
LIN {X -50.835,Y -100.986,Z 121,A -120.8979,B 24.9546,C -1.5568,E1 24.9271,E2 206.8863} C_DIS
LIN {X -53.6019,Y -99.5432,Z 121,A -122.4371,B 24.9544,C -1.5607,E1 24.9233,E2 208.4207} C_DIS
LIN {X -57.4926,Y -97.3473,Z 121,A -124.6209,B 24.954,C -1.5672,E1 24.918,E2 210.5955} C_DIS
LIN {X -60.2934,Y -95.639,Z 121,A -126.4384,B 24.9542,C -1.5634,E1 24.9136,E2 212.4277} C_DIS
LIN {X -62.8249,Y -93.9967,Z 121,A -127.9539,B 24.954,C -1.5664,E1 24.9101,E2 213.9411} C_DIS
LIN {X -65.3855,Y -92.232,Z 121,A -129.4106,B 24.9536,C -1.5739,E1 24.9068,E2 215.3848} C_DIS
LIN {X -67.6248,Y -90.603,Z 121,A -130.9017,B 24.9536,C -1.5728,E1 24.9034,E2 216.8839} C_DIS
LIN {X -70.2347,Y -88.5946,Z 121,A -132.5732,B 24.9535,C -1.5757,E1 24.8998,E2 218.5546} C_DIS
LIN {X -72.9294,Y -86.3913,Z 121,A -134.2653,B 24.9531,C -1.582,E1 24.8962,E2 220.2382} C_DIS
LIN {X -75.0211,Y -84.5813,Z 121,A -135.7873,B 24.9532,C -1.5799,E1 24.8929,E2 221.7712} C_DIS
LIN {X -77.4486,Y -82.3626,Z 121,A -137.3482,B 24.9528,C -1.5876,E1 24.8898,E2 223.3201} C_DIS
LIN {X -79.4537,Y -80.4301,Z 121,A -138.7663,B 24.9526,C -1.5903,E1 24.8869,E2 224.7377} C_DIS
LIN {X -81.5953,Y -78.2571,Z 121,A -140.3734,B 24.9526,C -1.5912,E1 24.8838,E2 226.3496} C_DIS
LIN {X -83.7287,Y -75.9723,Z 121,A -141.9878,B 24.9524,C -1.5935,E1 24.8807,E2 227.9656} C_DIS
LIN {X -85.7241,Y -73.7125,Z 121,A -143.5596,B 24.9524,C -1.5953,E1 24.8778,E2 229.5403} C_DIS
LIN {X -87.8307,Y -71.1875,Z 121,A -145.1574,B 24.9519,C -1.602,E1 24.875,E2 231.1294} C_DIS
LIN {X -89.9807,Y -68.4532,Z 121,A -146.8934,B 24.9516,C -1.6073,E1 24.8721,E2 232.8611} C_DIS
LIN {X -91.6302,Y -66.229,Z 121,A -148.4734,B 24.9518,C -1.6038,E1 24.8694,E2 234.4571} C_DIS
LIN {X -93.5064,Y -63.5491,Z 121,A -149.8155,B 24.9508,C -1.6206,E1 24.8674,E2 235.7658} C_DIS
LIN {X -94.993,Y -61.3049,Z 121,A -151.3359,B 24.9509,C -1.618,E1 24.865,E2 237.3002} C_DIS
LIN {X -96.2681,Y -59.2857,Z 121,A -152.7367,B 24.9512,C -1.6136,E1 24.8629,E2 238.7186} C_DIS
LIN {X -97.8564,Y -56.6227,Z 121,A -154.1416,B 24.9506,C -1.6244,E1 24.861,E2 240.1048} C_DIS
LIN {X -99.0512,Y -54.5089,Z 121,A -155.3789,B 24.9504,C -1.6275,E1 24.8593,E2 241.3414} C_DIS
LIN {X -100.5118,Y -51.7629,Z 121,A -156.8072,B 24.9497,C -1.6377,E1 24.8574,E2 242.7529} C_DIS
LIN {X -101.8051,Y -49.1698,Z 121,A -158.2307,B 24.9494,C -1.6437,E1 24.8557,E2 244.1699} C_DIS
LIN {X -102.8185,Y -47.0174,Z 121,A -159.7707,B 24.95,C -1.6339,E1 24.8538,E2 245.7416} C_DIS
LIN {X -104.0585,Y -44.2022,Z 121,A -161.2533,B 24.9495,C -1.6414,E1 24.8522,E2 247.2144} C_DIS
LIN {X -105.1011,Y -41.6627,Z 121,A -162.6206,B 24.9492,C -1.6464,E1 24.8508,E2 248.5774} C_DIS
LIN {X -106.452,Y -38.0833,Z 121,A -164.576,B 24.9489,C -1.6515,E1 24.8489,E2 250.5317} C_DIS
LIN {X -107.4578,Y -35.1402,Z 121,A -166.0055,B 24.9482,C -1.6621,E1 24.8476,E2 251.9442} C_DIS
LIN {X -108.301,Y -32.4482,Z 121,A -167.6185,B 24.9484,C -1.6592,E1 24.8463,E2 253.5733} C_DIS
LIN {X -109.1244,Y -29.5595,Z 121,A -169.0489,B 24.9479,C -1.6675,E1 24.8452,E2 254.9923} C_DIS
LIN {X -110.0765,Y -25.791,Z 121,A -170.9603,B 24.9474,C -1.6759,E1 24.8439,E2 256.8948} C_DIS
LIN {X -110.6069,Y -23.4199,Z 121,A -172.4865,B 24.9479,C -1.6682,E1 24.843,E2 258.4484} C_DIS
LIN {X -111.1493,Y -20.6929,Z 121,A -173.9091,B 24.9476,C -1.6721,E1 24.8423,E2 259.8701} C_DIS
LIN {X -111.6258,Y -17.9453,Z 121,A -175.3402,B 24.9474,C -1.6759,E1 24.8416,E2 261.3007} C_DIS
LIN {X -112.0749,Y -14.8736,Z 121,A -176.6784,B 24.9465,C -1.6901,E1 24.8411,E2 262.613} C_DIS
LIN {X -112.42,Y -11.9864,Z 121,A -178.0727,B 24.946,C -1.6979,E1 24.8407,E2 263.9969} C_DIS
LIN {X -112.6719,Y -9.3298,Z 121,A -179.4723,B 24.9458,C -1.7004,E1 24.8403,E2 265.399} C_DIS
LIN {X -112.8662,Y -6.5753,Z 121,A 178.9633,B 24.9459,C -1.6985,E1 24.84,E2 266.9774} C_DIS
LIN {X -113.0251,Y -2.7746,Z 121,A 177.0199,B 24.9456,C -1.7041,E1 24.8398,E2 268.9191} C_DIS
LIN {X -113.0584,Y 0.1353,Z 121,A 175.4622,B 24.9455,C -1.7057,E1 24.8398,E2 270.4825} C_DIS
LIN {X -113.0145,Y 3.1189,Z 121,A 174.1494,B 24.9447,C -1.7184,E1 24.8398,E2 271.7729} C_DIS
LIN {X -112.9215,Y 5.5747,Z 121,A 172.6357,B 24.9451,C -1.712,E1 24.8401,E2 273.3109} C_DIS
LIN {X -112.752,Y 8.3274,Z 121,A 171.2264,B 24.9448,C -1.7161,E1 24.8403,E2 274.719} C_DIS
LIN {X -112.48,Y 11.4139,Z 121,A 169.7576,B 24.9442,C -1.7251,E1 24.8407,E2 276.1749} C_DIS
LIN {X -112.2064,Y 13.8592,Z 121,A 168.3887,B 24.9442,C -1.7244,E1 24.8412,E2 277.5537} C_DIS
LIN {X -111.7816,Y 16.9376,Z 121,A 167.0853,B 24.9433,C -1.7401,E1 24.8417,E2 278.8275} C_DIS
LIN {X -111.3336,Y 19.6684,Z 121,A 165.6739,B 24.943,C -1.7443,E1 24.8423,E2 280.2373} C_DIS
LIN {X -110.8188,Y 22.3877,Z 121,A 164.1031,B 24.9431,C -1.7423,E1 24.8432,E2 281.8221} C_DIS
LIN {X -110.3142,Y 24.7614,Z 121,A 162.7045,B 24.9433,C -1.7397,E1 24.844,E2 283.2353} C_DIS
LIN {X -109.6696,Y 27.4765,Z 121,A 161.4408,B 24.9426,C -1.75,E1 24.8448,E2 284.4817} C_DIS
LIN {X -108.848,Y 30.5627,Z 121,A 159.7874,B 24.9423,C -1.7539,E1 24.8461,E2 286.1354} C_DIS
LIN {X -108.0734,Y 33.1983,Z 121,A 158.5637,B 24.9416,C -1.7649,E1 24.847,E2 287.34} C_DIS
LIN {X -107.2334,Y 35.8189,Z 121,A 157.0014,B 24.9418,C -1.7627,E1 24.8484,E2 288.9164} C_DIS
LIN {X -106.4447,Y 38.1036,Z 121,A 155.7743,B 24.9415,C -1.7664,E1 24.8495,E2 290.1416} C_DIS
LIN {X -105.4703,Y 40.7228,Z 121,A 154.3612,B 24.9412,C -1.771,E1 24.8509,E2 291.5518} C_DIS
LIN {X -104.4596,Y 43.2497,Z 121,A 152.9531,B 24.941,C -1.7741,E1 24.8524,E2 292.9603} C_DIS
LIN {X -103.219,Y 46.1287,Z 121,A 151.3579,B 24.9407,C -1.7787,E1 24.8542,E2 294.5532} C_DIS
LIN {X -102.0308,Y 48.7,Z 121,A 149.9308,B 24.9404,C -1.7834,E1 24.8559,E2 295.977} C_DIS
LIN {X -100.822,Y 51.1559,Z 121,A 148.5231,B 24.9402,C -1.7868,E1 24.8576,E2 297.3843} C_DIS
LIN {X -99.548,Y 53.593,Z 121,A 147.2697,B 24.9395,C -1.7964,E1 24.8592,E2 298.6214} C_DIS
LIN {X -98.1612,Y 56.0923,Z 121,A 145.5885,B 24.9398,C -1.7915,E1 24.8616,E2 300.323} C_DIS
LIN {X -96.2463,Y 59.3212,Z 121,A 143.7434,B 24.9393,C -1.7992,E1 24.8642,E2 302.1592} C_DIS
LIN {X -94.5812,Y 61.9387,Z 121,A 142.3166,B 24.9386,C -1.8094,E1 24.8663,E2 303.5689} C_DIS
LIN {X -93.04,Y 64.2307,Z 121,A 140.7527,B 24.9388,C -1.8069,E1 24.8688,E2 305.1466} C_DIS
LIN {X -91.444,Y 66.4833,Z 121,A 139.3458,B 24.9386,C -1.8105,E1 24.8711,E2 306.5519} C_DIS
LIN {X -89.153,Y 69.5274,Z 121,A 137.1925,B 24.9388,C -1.8069,E1 24.8748,E2 308.7238} C_DIS
LIN {X -86.8361,Y 72.3976,Z 121,A 135.4526,B 24.9381,C -1.817,E1 24.8778,E2 310.4479} C_DIS
LIN {X -84.5789,Y 75.0238,Z 121,A 133.6431,B 24.938,C -1.8193,E1 24.8812,E2 312.2599} C_DIS
LIN {X -82.3582,Y 77.4533,Z 121,A 132.079,B 24.9374,C -1.8277,E1 24.8841,E2 313.8112} C_DIS
LIN {X -80.4357,Y 79.448,Z 121,A 130.6241,B 24.9373,C -1.8291,E1 24.8869,E2 315.2688} C_DIS
LIN {X -77.9515,Y 81.8897,Z 121,A 128.7193,B 24.9373,C -1.8278,E1 24.8908,E2 317.1847} C_DIS
LIN {X -75.4072,Y 84.2357,Z 121,A 127.1302,B 24.9366,C -1.8385,E1 24.894,E2 318.7548} C_DIS
LIN {X -73.3205,Y 86.0581,Z 121,A 125.7191,B 24.9364,C -1.8414,E1 24.897,E2 320.1645} C_DIS
LIN {X -71.1899,Y 87.8288,Z 121,A 124.2508,B 24.9364,C -1.8419,E1 24.9002,E2 321.637} C_DIS
LIN {X -68.358,Y 90.0522,Z 121,A 122.4874,B 24.936,C -1.8483,E1 24.9041,E2 323.3918} C_DIS
LIN {X -66.1704,Y 91.672,Z 121,A 121.097,B 24.9358,C -1.8507,E1 24.9072,E2 324.7813} C_DIS
LIN {X -63.6479,Y 93.4395,Z 121,A 119.6799,B 24.9352,C -1.8596,E1 24.9104,E2 326.182} C_DIS
LIN {X -61.2974,Y 94.9979,Z 121,A 118.1005,B 24.9354,C -1.8564,E1 24.9141,E2 327.7742} C_DIS
LIN {X -59.3179,Y 96.2483,Z 121,A 116.7605,B 24.9357,C -1.8524,E1 24.9173,E2 329.1278} C_DIS
LIN {X -56.6166,Y 97.8599,Z 121,A 115.2955,B 24.9351,C -1.8605,E1 24.9208,E2 330.5781} C_DIS
LIN {X -54.5043,Y 99.0537,Z 121,A 114.0615,B 24.935,C -1.8625,E1 24.9238,E2 331.8109} C_DIS
LIN {X -51.7599,Y 100.5133,Z 121,A 112.6377,B 24.9344,C -1.8713,E1 24.9273,E2 333.2177} C_DIS
LIN {X -49.2546,Y 101.7643,Z 121,A 111.2121,B 24.9342,C -1.8733,E1 24.9309,E2 334.6423} C_DIS
LIN {X -47.0671,Y 102.7961,Z 121,A 109.7023,B 24.9349,C -1.8637,E1 24.9348,E2 336.1788} C_DIS
LIN {X -44.231,Y 104.0463,Z 121,A 108.2517,B 24.9344,C -1.8709,E1 24.9384,E2 337.6156} C_DIS
LIN {X -41.6785,Y 105.0949,Z 121,A 106.8492,B 24.9343,C -1.8727,E1 24.9421,E2 339.017} C_DIS
LIN {X -39.421,Y 105.9637,Z 121,A 105.6069,B 24.9342,C -1.8736,E1 24.9453,E2 340.2597} C_DIS
LIN {X -36.7621,Y 106.9154,Z 121,A 104.058,B 24.9344,C -1.8706,E1 24.9494,E2 341.8187} C_DIS
LIN {X -34.1332,Y 107.7835,Z 121,A 102.7764,B 24.9339,C -1.8772,E1 24.9528,E2 343.0869} C_DIS
LIN {X -31.1553,Y 108.6801,Z 121,A 101.1963,B 24.9339,C -1.8788,E1 24.957,E2 344.6658} C_DIS
LIN {X -28.4211,Y 109.4268,Z 121,A 99.9095,B 24.9333,C -1.8864,E1 24.9605,E2 345.9365} C_DIS
LIN {X -25.7494,Y 110.0861,Z 121,A 98.5139,B 24.9332,C -1.8877,E1 24.9642,E2 347.3309} C_DIS
LIN {X -23.3899,Y 110.6131,Z 121,A 97.0092,B 24.9339,C -1.8773,E1 24.9684,E2 348.8623} C_DIS
LIN {X -20.6828,Y 111.1512,Z 121,A 95.6065,B 24.9339,C -1.8782,E1 24.9723,E2 350.2643} C_DIS
LIN {X -17.9623,Y 111.6231,Z 121,A 94.3278,B 24.9334,C -1.8842,E1 24.9758,E2 351.53} C_DIS
LIN {X -14.8946,Y 112.0722,Z 121,A 92.9036,B 24.9329,C -1.8914,E1 24.9796,E2 352.9383} C_DIS
LIN {X -12.4926,Y 112.3667,Z 121,A 91.5267,B 24.9333,C -1.8858,E1 24.9835,E2 354.3294} C_DIS
LIN {X -9.7377,Y 112.6388,Z 121,A 89.862,B 24.9341,C -1.8756,E1 24.9882,E2 356.0191} C_DIS
LIN {X -5.2421,Y 112.9361,Z 121,A 87.8912,B 24.9331,C -1.8895,E1 24.9936,E2 357.9574} C_DIS
LIN {X -2.6888,Y 113.0267,Z 121,A 86.4389,B 24.9335,C -1.8833,E1 24.9977,E2 359.4247} C_DIS
LIN {X 0.4167,Y 113.0566,Z 121,A 84.9743,B 24.9332,C -1.8882,E1 25.0018,E2 360.8776} C_DIS
LIN {X 3.1469,Y 113.0137,Z 121,A 83.5205,B 24.9334,C -1.8854,E1 25.0058,E2 362.3378} C_DIS
LIN {X 5.7391,Y 112.9124,Z 121,A 82.1803,B 24.9334,C -1.8844,E1 25.0096,E2 363.6799} C_DIS
LIN {X 8.4048,Y 112.7458,Z 121,A 80.8023,B 24.9335,C -1.8833,E1 25.0134,E2 365.0599} C_DIS
LIN {X 11.4688,Y 112.4742,Z 121,A 79.36,B 24.9332,C -1.8881,E1 25.0174,E2 366.49} C_DIS
LIN {X 13.8632,Y 112.2058,Z 121,A 77.9698,B 24.9337,C -1.8807,E1 25.0213,E2 367.8967} C_DIS
LIN {X 16.9246,Y 111.7836,Z 121,A 76.7147,B 24.9328,C -1.8935,E1 25.0247,E2 369.1204} C_DIS
LIN {X 19.6766,Y 111.3321,Z 121,A 75.3152,B 24.9328,C -1.8935,E1 25.0285,E2 370.5183} C_DIS
LIN {X 22.5171,Y 110.7923,Z 121,A 73.7322,B 24.9332,C -1.8879,E1 25.0329,E2 372.1128} C_DIS
LIN {X 24.78,Y 110.3101,Z 121,A 72.3979,B 24.9337,C -1.8804,E1 25.0366,E2 373.4631} C_DIS
LIN {X 27.4735,Y 109.6703,Z 121,A 71.1219,B 24.9334,C -1.885,E1 25.04,E2 374.7264} C_DIS
LIN {X 30.1505,Y 108.9647,Z 121,A 69.5905,B 24.9338,C -1.8786,E1 25.0442,E2 376.2705} C_DIS
LIN {X 33.1529,Y 108.0874,Z 121,A 68.0517,B 24.9338,C -1.8794,E1 25.0483,E2 377.8047} C_DIS
LIN {X 35.8763,Y 107.214,Z 121,A 66.7199,B 24.9335,C -1.8833,E1 25.0518,E2 379.1248} C_DIS
LIN {X 38.0911,Y 106.4492,Z 121,A 65.5063,B 24.9337,C -1.881,E1 25.055,E2 380.3413} C_DIS
LIN {X 40.6869,Y 105.4844,Z 121,A 64.1046,B 24.9337,C -1.8797,E1 25.0586,E2 381.743} C_DIS
LIN {X 43.7957,Y 104.2298,Z 121,A 62.6597,B 24.9331,C -1.889,E1 25.0623,E2 383.1626} C_DIS
LIN {X 46.1378,Y 103.2149,Z 121,A 61.1207,B 24.934,C -1.8769,E1 25.0663,E2 384.7266} C_DIS
LIN {X 48.3408,Y 102.2034,Z 121,A 59.7661,B 24.9345,C -1.8699,E1 25.0698,E2 386.0942} C_DIS
LIN {X 50.8376,Y 100.9847,Z 121,A 58.3647,B 24.9345,C -1.8684,E1 25.0733,E2 387.4954} C_DIS
LIN {X 53.5963,Y 99.5463,Z 121,A 57.0741,B 24.9338,C -1.8788,E1 25.0764,E2 388.7578} C_DIS
LIN {X 55.7227,Y 98.3735,Z 121,A 55.6903,B 24.9344,C -1.8703,E1 25.0798,E2 390.1576} C_DIS
LIN {X 58.4073,Y 96.8019,Z 121,A 54.0276,B 24.9349,C -1.8642,E1 25.0838,E2 391.8296} C_DIS
LIN {X 61.9505,Y 94.5735,Z 121,A 52.1607,B 24.9343,C -1.872,E1 25.0882,E2 393.672} C_DIS
LIN {X 64.2479,Y 93.028,Z 121,A 50.6074,B 24.9349,C -1.8631,E1 25.0918,E2 395.2412} C_DIS
LIN {X 66.6194,Y 91.3444,Z 121,A 49.1854,B 24.9349,C -1.8628,E1 25.095,E2 396.6587} C_DIS
LIN {X 68.8627,Y 89.6652,Z 121,A 47.6721,B 24.9354,C -1.8562,E1 25.0984,E2 398.1824} C_DIS
LIN {X 71.3273,Y 87.7174,Z 121,A 46.0729,B 24.9356,C -1.8528,E1 25.1019,E2 399.7835} C_DIS
LIN {X 73.973,Y 85.4995,Z 121,A 44.3982,B 24.9356,C -1.8528,E1 25.1054,E2 401.4519} C_DIS
LIN {X 76.3163,Y 83.4131,Z 121,A 42.7698,B 24.936,C -1.8478,E1 25.1088,E2 403.0853} C_DIS
LIN {X 78.4597,Y 81.4001,Z 121,A 41.2746,B 24.9362,C -1.8445,E1 25.1119,E2 404.5823} C_DIS
LIN {X 81.0674,Y 78.8048,Z 121,A 39.3678,B 24.9366,C -1.8385,E1 25.1156,E2 406.495} C_DIS
LIN {X 83.3127,Y 76.4257,Z 121,A 37.8243,B 24.9366,C -1.8399,E1 25.1185,E2 408.0284} C_DIS
LIN {X 85.1539,Y 74.3687,Z 121,A 36.4324,B 24.9367,C -1.837,E1 25.1211,E2 409.421} C_DIS
LIN {X 86.9591,Y 72.2496,Z 121,A 35.0275,B 24.937,C -1.8339,E1 25.1236,E2 410.8267} C_DIS
LIN {X 88.8087,Y 69.9638,Z 121,A 33.4792,B 24.9374,C -1.8277,E1 25.1263,E2 412.3824} C_DIS
LIN {X 90.8093,Y 67.3502,Z 121,A 31.8855,B 24.9374,C -1.8269,E1 25.129,E2 413.9705} C_DIS
LIN {X 92.431,Y 65.1067,Z 121,A 30.368,B 24.938,C -1.8182,E1 25.1315,E2 415.5011} C_DIS
LIN {X 93.9972,Y 62.8242,Z 121,A 28.969,B 24.9383,C -1.8147,E1 25.1337,E2 416.9014} C_DIS
LIN {X 95.8324,Y 59.9839,Z 121,A 27.3524,B 24.9383,C -1.8147,E1 25.1361,E2 418.5101} C_DIS
LIN {X 97.153,Y 57.8213,Z 121,A 26.1149,B 24.9383,C -1.8133,E1 25.1379,E2 419.7445} C_DIS
LIN {X 98.5399,Y 55.4248,Z 121,A 24.8759,B 24.9381,C -1.8169,E1 25.1396,E2 420.9685} C_DIS
LIN {X 99.7089,Y 53.2965,Z 121,A 23.3642,B 24.9392,C -1.8007,E1 25.1416,E2 422.5104} C_DIS
LIN {X 100.9932,Y 50.8205,Z 121,A 21.9294,B 24.9396,C -1.7958,E1 25.1434,E2 423.9492} C_DIS
LIN {X 102.2029,Y 48.3418,Z 121,A 20.7013,B 24.9393,C -1.7995,E1 25.1449,E2 425.1621} C_DIS
LIN {X 103.4957,Y 45.5046,Z 121,A 19.0483,B 24.9398,C -1.7917,E1 25.1468,E2 426.8245} C_DIS
LIN {X 104.7583,Y 42.516,Z 121,A 17.4177,B 24.9401,C -1.7875,E1 25.1485,E2 428.456} C_DIS
LIN {X 106.0925,Y 39.069,Z 121,A 15.7927,B 24.9397,C -1.7932,E1 25.1501,E2 430.0584} C_DIS
LIN {X 106.9087,Y 36.7819,Z 121,A 14.2645,B 24.9409,C -1.7759,E1 25.1516,E2 431.6189} C_DIS
LIN {X 107.7868,Y 34.1226,Z 121,A 13.0052,B 24.9407,C -1.7789,E1 25.1526,E2 432.864} C_DIS
LIN {X 108.6819,Y 31.1489,Z 121,A 11.3732,B 24.9412,C -1.7714,E1 25.1539,E2 434.5043} C_DIS
LIN {X 109.6709,Y 27.4714,Z 121,A 9.3768,B 24.9418,C -1.7624,E1 25.1553,E2 436.5105} C_DIS
LIN {X 110.3172,Y 24.7478,Z 121,A 8.1178,B 24.9416,C -1.7652,E1 25.1561,E2 437.7554} C_DIS
LIN {X 110.9849,Y 21.5469,Z 121,A 6.7043,B 24.9412,C -1.7712,E1 25.1569,E2 439.1466} C_DIS
LIN {X 111.4477,Y 19.0114,Z 121,A 5.3167,B 24.9417,C -1.7633,E1 25.1576,E2 440.5446} C_DIS
LIN {X 111.8295,Y 16.6281,Z 121,A 3.824,B 24.9428,C -1.747,E1 25.1582,E2 442.067} C_DIS
LIN {X 112.2101,Y 13.8296,Z 121,A 2.5346,B 24.9427,C -1.749,E1 25.1587,E2 443.3443} C_DIS
LIN {X 112.5152,Y 11.0772,Z 121,A 1.0158,B 24.9433,C -1.7391,E1 25.1591,E2 444.8772} C_DIS
LIN {X 112.7527,Y 8.3181,Z 121,A -0.3782,B 24.9436,C -1.735,E1 25.1594,E2 446.2727} C_DIS
LIN {X 112.9374,Y 5.2118,Z 121,A -1.9112,B 24.9438,C -1.732,E1 25.1597,E2 447.8038} C_DIS
LIN {X 113.0507,Y 1.3833,Z 121,A -3.8033,B 24.944,C -1.7279,E1 25.1597,E2 449.6942} C_DIS
LIN {X 113.0444,Y -1.7281,Z 121,A -5.3134,B 24.9442,C -1.7258,E1 25.1597,E2 451.2002} C_DIS
LIN {X 112.9827,Y -4.1569,Z 121,A -6.5364,B 24.9444,C -1.7222,E1 25.1597,E2 452.4246} C_DIS
LIN {X 112.824,Y -7.2637,Z 121,A -8.1684,B 24.9449,C -1.7145,E1 25.1594,E2 454.0649} C_DIS
LIN {X 112.5853,Y -10.3178,Z 121,A -9.6203,B 24.9449,C -1.714,E1 25.159,E2 455.5092} C_DIS
LIN {X 112.3149,Y -12.9345,Z 121,A -10.8139,B 24.9449,C -1.7161,E1 25.1587,E2 456.6909} C_DIS
LIN {X 111.9728,Y -15.6223,Z 121,A -12.324,B 24.9455,C -1.7053,E1 25.1581,E2 458.2176} C_DIS
LIN {X 111.6181,Y -17.9923,Z 121,A -13.6532,B 24.9461,C -1.6961,E1 25.1576,E2 459.5608} C_DIS
LIN {X 111.1494,Y -20.6926,Z 121,A -15.0488,B 24.9464,C -1.6912,E1 25.1569,E2 460.9596} C_DIS
LIN {X 110.5307,Y -23.7689,Z 121,A -16.3409,B 24.9459,C -1.6999,E1 25.1561,E2 462.2238} C_DIS
LIN {X 109.916,Y -26.4667,Z 121,A -17.7325,B 24.9461,C -1.6958,E1 25.1553,E2 463.6169} C_DIS
LIN {X 109.3241,Y -28.8203,Z 121,A -19.1082,B 24.9468,C -1.6851,E1 25.1543,E2 465.0099} C_DIS
LIN {X 108.489,Y -31.8145,Z 121,A -20.6733,B 24.9471,C -1.6806,E1 25.1531,E2 466.5767} C_DIS
LIN {X 107.7825,Y -34.1364,Z 121,A -22.0177,B 24.9477,C -1.6714,E1 25.152,E2 467.9351} C_DIS
LIN {X 106.8021,Y -37.0854,Z 121,A -23.312,B 24.9472,C -1.6793,E1 25.1508,E2 469.2034} C_DIS
LIN {X 105.7939,Y -39.8696,Z 121,A -24.9901,B 24.948,C -1.6665,E1 25.1492,E2 470.9025} C_DIS
LIN {X 104.5297,Y -43.0776,Z 121,A -26.7267,B 24.9483,C -1.6615,E1 25.1474,E2 472.6412} C_DIS
LIN {X 103.212,Y -46.1443,Z 121,A -28.3691,B 24.9485,C -1.6586,E1 25.1456,E2 474.2815} C_DIS
LIN {X 102.1962,Y -48.3557,Z 121,A -29.7142,B 24.949,C -1.6497,E1 25.1439,E2 475.6404} C_DIS
LIN {X 100.9839,Y -50.8391,Z 121,A -31.1068,B 24.9492,C -1.6458,E1 25.1422,E2 477.0346} C_DIS
LIN {X 99.5488,Y -53.5916,Z 121,A -32.3935,B 24.9487,C -1.6543,E1 25.1406,E2 478.2946} C_DIS
LIN {X 98.3785,Y -55.7138,Z 121,A -33.7676,B 24.9494,C -1.6439,E1 25.1387,E2 479.6859} C_DIS
LIN {X 96.8119,Y -58.3909,Z 121,A -35.409,B 24.9498,C -1.6362,E1 25.1363,E2 481.3372} C_DIS
LIN {X 94.5824,Y -61.9369,Z 121,A -37.5332,B 24.9502,C -1.63,E1 25.1331,E2 483.4652} C_DIS
LIN {X 93.0258,Y -64.2511,Z 121,A -38.8436,B 24.9502,C -1.6307,E1 25.1311,E2 484.7674} C_DIS
LIN {X 91.4244,Y -66.5101,Z 121,A -40.2387,B 24.9504,C -1.6272,E1 25.1288,E2 486.1641} C_DIS
LIN {X 89.872,Y -68.5943,Z 121,A -41.6607,B 24.9509,C -1.6188,E1 25.1264,E2 487.5992} C_DIS
LIN {X 87.8309,Y -71.1873,Z 121,A -43.246,B 24.9509,C -1.6183,E1 25.1236,E2 489.1783} C_DIS
LIN {X 85.6027,Y -73.8549,Z 121,A -45.0309,B 24.9513,C -1.6126,E1 25.1204,E2 490.9686} C_DIS
LIN {X 83.4159,Y -76.3132,Z 121,A -46.6642,B 24.9514,C -1.6098,E1 25.1173,E2 492.601} C_DIS
LIN {X 81.4029,Y -78.4567,Z 121,A -48.1032,B 24.9515,C -1.6084,E1 25.1146,E2 494.0371} C_DIS
LIN {X 79.4422,Y -80.4415,Z 121,A -49.5441,B 24.9518,C -1.6037,E1 25.1117,E2 495.483} C_DIS
LIN {X 76.9421,Y -82.8388,Z 121,A -51.4283,B 24.9524,C -1.5936,E1 25.1079,E2 497.3833} C_DIS
LIN {X 74.3693,Y -85.1534,Z 121,A -53.0013,B 24.9522,C -1.5977,E1 25.1046,E2 498.9403} C_DIS
LIN {X 72.2607,Y -86.9499,Z 121,A -54.4409,B 24.9525,C -1.5929,E1 25.1015,E2 500.3857} C_DIS
LIN {X 69.5502,Y -89.1355,Z 121,A -56.1537,B 24.9525,C -1.5913,E1 25.0978,E2 502.0959} C_DIS
LIN {X 67.3141,Y -90.8357,Z 121,A -57.5533,B 24.9527,C -1.5894,E1 25.0947,E2 503.4951} C_DIS
LIN {X 65.1004,Y -92.4355,Z 121,A -59.0747,B 24.9532,C -1.5803,E1 25.0912,E2 505.0326} C_DIS
LIN {X 62.8168,Y -94.0022,Z 121,A -60.4703,B 24.9534,C -1.5778,E1 25.0879,E2 506.4294} C_DIS
LIN {X 59.9339,Y -95.8636,Z 121,A -62.1294,B 24.9534,C -1.5781,E1 25.084,E2 508.0825} C_DIS
LIN {X 56.8739,Y -97.7121,Z 121,A -63.9996,B 24.9537,C -1.5721,E1 25.0795,E2 509.9612} C_DIS
LIN {X 53.2675,Y -99.7241,Z 121,A -66.0888,B 24.9539,C -1.5685,E1 25.0744,E2 512.0527} C_DIS
LIN {X 50.8186,Y -100.9942,Z 121,A -67.4834,B 24.954,C -1.5663,E1 25.0709,E2 513.4487} C_DIS
LIN {X 47.0869,Y -102.7871,Z 121,A -69.5741,B 24.9542,C -1.5633,E1 25.0656,E2 515.5412} C_DIS
LIN {X 44.2515,Y -104.0377,Z 121,A -71.0615,B 24.9542,C -1.5646,E1 25.0618,E2 517.0218} C_DIS
LIN {X 41.6558,Y -105.1038,Z 121,A -72.4353,B 24.9542,C -1.5647,E1 25.0583,E2 518.3922} C_DIS
LIN {X 39.069,Y -106.0925,Z 121,A -73.6778,B 24.9538,C -1.5699,E1 25.0551,E2 519.6197} C_DIS
LIN {X 36.2741,Y -107.0799,Z 121,A -75.3554,B 24.9544,C -1.5603,E1 25.0506,E2 521.3169} C_DIS
LIN {X 32.2358,Y -108.364,Z 121,A -77.3967,B 24.9543,C -1.5624,E1 25.0452,E2 523.3495} C_DIS
LIN {X 29.8134,Y -109.0558,Z 121,A -78.748,B 24.9545,C -1.5577,E1 25.0415,E2 524.7097} C_DIS
LIN {X 27.467,Y -109.6719,Z 121,A -80.1082,B 24.9549,C -1.5506,E1 25.0378,E2 526.0845} C_DIS
LIN {X 24.466,Y -110.3787,Z 121,A -81.4921,B 24.9546,C -1.557,E1 25.0341,E2 527.4515} C_DIS
LIN {X 21.5933,Y -110.976,Z 121,A -82.8632,B 24.9544,C -1.5608,E1 25.0304,E2 528.812} C_DIS
LIN {X 18.9341,Y -111.4607,Z 121,A -84.2275,B 24.9544,C -1.5599,E1 25.0266,E2 530.1768} C_DIS
LIN {X 16.4645,Y -111.8532,Z 121,A -85.7266,B 24.9551,C -1.5489,E1 25.0224,E2 531.7006} C_DIS
LIN {X 13.8681,Y -112.2052,Z 121,A -86.9786,B 24.9549,C -1.5513,E1 25.019,E2 532.9458} C_DIS
LIN {X 11.0716,Y -112.5157,Z 121,A -88.5267,B 24.9553,C -1.5452,E1 25.0146,E2 534.5074} C_DIS
LIN {X 8.3126,Y -112.7531,Z 121,A -89.9292,B 24.9553,C -1.5445,E1 25.0107,E2 535.9108} C_DIS
LIN {X 5.2071,Y -112.9376,Z 121,A -91.4369,B 24.9552,C -1.5469,E1 25.0065,E2 537.4123} C_DIS
LIN {X 1.3791,Y -113.0507,Z 121,A -93.4438,B 24.9554,C -1.5434,E1 25.0009,E2 539.427} C_DIS
LIN {X 1.3791,Y -113.0507,Z 121,A -93.4438,B 24.9554,C -1.5434,E1 25.0009,E2 539.427} C_DIS
Enddeposition()
LIN {X 0.8387,Y -118.9462,Z 122,A -93.1377,B 24.9593,C -1.4737,E1 25.0013,E2 539.2863} C_DIS
Startdeposition()
$VEL.CP = VEL_PRINT
LIN {X 2.9192,Y -118.9156,Z 122,A -91.7713,B 24.9584,C -1.4907,E1 25.0052,E2 537.8797} C_DIS
LIN {X 5.8367,Y -118.8081,Z 122,A -90.3663,B 24.9584,C -1.4912,E1 25.0091,E2 536.474} C_DIS
LIN {X 8.7506,Y -118.6291,Z 122,A -88.8057,B 24.9579,C -1.499,E1 25.0135,E2 534.8955} C_DIS
LIN {X 12.2551,Y -118.3162,Z 122,A -87.2685,B 24.9583,C -1.4926,E1 25.0178,E2 533.3744} C_DIS
LIN {X 16.0086,Y -117.8693,Z 122,A -85.45,B 24.9583,C -1.4937,E1 25.0228,E2 531.555} C_DIS
LIN {X 18.8964,Y -117.4409,Z 122,A -84.0462,B 24.9582,C -1.4946,E1 25.0267,E2 530.1503} C_DIS
LIN {X 21.7728,Y -116.9418,Z 122,A -82.6423,B 24.9581,C -1.4956,E1 25.0306,E2 528.7455} C_DIS
LIN {X 24.6362,Y -116.3722,Z 122,A -81.2388,B 24.9581,C -1.4967,E1 25.0344,E2 527.3411} C_DIS
LIN {X 27.4847,Y -115.7326,Z 122,A -79.8354,B 24.958,C -1.4979,E1 25.0382,E2 525.9368} C_DIS
LIN {X 30.3166,Y -115.0232,Z 122,A -78.4322,B 24.9579,C -1.4993,E1 25.042,E2 524.5326} C_DIS
LIN {X 33.1303,Y -114.2446,Z 122,A -77.0293,B 24.9579,C -1.5007,E1 25.0458,E2 523.1287} C_DIS
LIN {X 35.924,Y -113.3971,Z 122,A -75.6265,B 24.9577,C -1.5022,E1 25.0495,E2 521.7248} C_DIS
LIN {X 38.6961,Y -112.4813,Z 122,A -74.2244,B 24.9577,C -1.5038,E1 25.0532,E2 520.3217} C_DIS
LIN {X 41.4449,Y -111.4978,Z 122,A -72.8218,B 24.9575,C -1.5055,E1 25.0569,E2 518.9181} C_DIS
LIN {X 44.3241,Y -110.3839,Z 122,A -71.412,B 24.9576,C -1.5039,E1 25.0606,E2 517.515} C_DIS
LIN {X 46.8659,Y -109.3299,Z 122,A -70.0181,B 24.9573,C -1.5091,E1 25.0642,E2 516.1122} C_DIS
LIN {X 49.5349,Y -108.1468,Z 122,A -68.6164,B 24.9573,C -1.5111,E1 25.0677,E2 514.7093} C_DIS
LIN {X 52.174,Y -106.8986,Z 122,A -67.2152,B 24.9571,C -1.5132,E1 25.0713,E2 513.3068} C_DIS
LIN {X 54.7817,Y -105.586,Z 122,A -65.8141,B 24.957,C -1.5153,E1 25.0748,E2 511.9046} C_DIS
LIN {X 57.3564,Y -104.2098,Z 122,A -64.413,B 24.9569,C -1.5175,E1 25.0782,E2 510.5023} C_DIS
LIN {X 59.8966,Y -102.7708,Z 122,A -63.0123,B 24.9567,C -1.5198,E1 25.0816,E2 509.1003} C_DIS
LIN {X 62.4007,Y -101.2699,Z 122,A -61.6117,B 24.9566,C -1.5222,E1 25.0849,E2 507.6984} C_DIS
LIN {X 64.8672,Y -99.708,Z 122,A -60.2112,B 24.9564,C -1.5247,E1 25.0882,E2 506.2966} C_DIS
LIN {X 67.2946,Y -98.086,Z 122,A -58.811,B 24.9563,C -1.5273,E1 25.0915,E2 504.8951} C_DIS
LIN {X 69.6815,Y -96.405,Z 122,A -57.4111,B 24.9561,C -1.5299,E1 25.0947,E2 503.4939} C_DIS
LIN {X 72.1439,Y -94.5754,Z 122,A -56.0042,B 24.9561,C -1.5297,E1 25.0978,E2 502.0926} C_DIS
LIN {X 74.3279,Y -92.8698,Z 122,A -54.6115,B 24.9558,C -1.5354,E1 25.1009,E2 500.6916} C_DIS
LIN {X 76.5847,Y -91.0177,Z 122,A -53.2121,B 24.9557,C -1.5382,E1 25.1039,E2 499.2908} C_DIS
LIN {X 79.2088,Y -88.7407,Z 122,A -51.7868,B 24.9561,C -1.5302,E1 25.1068,E2 497.8902} C_DIS
LIN {X 80.9584,Y -87.1502,Z 122,A -50.4136,B 24.9553,C -1.5442,E1 25.1097,E2 496.4895} C_DIS
LIN {X 83.0728,Y -85.1372,Z 122,A -49.0148,B 24.9551,C -1.5472,E1 25.1125,E2 495.0893} C_DIS
LIN {X 85.1372,Y -83.0728,Z 122,A -47.6158,B 24.955,C -1.5504,E1 25.1153,E2 493.6888} C_DIS
LIN {X 87.5262,Y -80.5488,Z 122,A -45.9397,B 24.9547,C -1.5548,E1 25.1185,E2 492.0097} C_DIS
LIN {X 90.0711,Y -77.6958,Z 122,A -44.1195,B 24.9545,C -1.5585,E1 25.1218,E2 490.1888} C_DIS
LIN {X 91.9507,Y -75.462,Z 122,A -42.7212,B 24.9543,C -1.5618,E1 25.1243,E2 488.7891} C_DIS
LIN {X 93.7749,Y -73.1827,Z 122,A -41.3231,B 24.9541,C -1.5652,E1 25.1267,E2 487.3895} C_DIS
LIN {X 95.5427,Y -70.8593,Z 122,A -39.9249,B 24.9539,C -1.5687,E1 25.1291,E2 485.9899} C_DIS
LIN {X 97.2529,Y -68.4932,Z 122,A -38.5271,B 24.9537,C -1.5722,E1 25.1313,E2 484.5905} C_DIS
LIN {X 98.9045,Y -66.0859,Z 122,A -37.1294,B 24.9535,C -1.5758,E1 25.1335,E2 483.1913} C_DIS
LIN {X 100.7069,Y -63.3019,Z 122,A -35.7129,B 24.9537,C -1.5716,E1 25.1357,E2 481.7919} C_DIS
LIN {X 102.028,Y -61.1532,Z 122,A -34.3339,B 24.953,C -1.5831,E1 25.1377,E2 480.3928} C_DIS
LIN {X 103.4981,Y -58.6309,Z 122,A -32.9365,B 24.9528,C -1.5868,E1 25.1396,E2 478.9939} C_DIS
LIN {X 104.9058,Y -56.0733,Z 122,A -31.5391,B 24.9526,C -1.5906,E1 25.1415,E2 477.5949} C_DIS
LIN {X 106.2503,Y -53.4819,Z 122,A -30.142,B 24.9524,C -1.5943,E1 25.1433,E2 476.1963} C_DIS
LIN {X 107.7135,Y -50.4657,Z 122,A -28.4925,B 24.952,C -1.601,E1 25.1453,E2 474.54} C_DIS
LIN {X 108.9859,Y -47.6549,Z 122,A -27.0611,B 24.9519,C -1.6029,E1 25.1469,E2 473.1119} C_DIS
LIN {X 110.1226,Y -44.9659,Z 122,A -25.6641,B 24.9516,C -1.6068,E1 25.1484,E2 471.7134} C_DIS
LIN {X 111.4978,Y -41.4449,Z 122,A -23.8553,B 24.9513,C -1.6119,E1 25.1502,E2 469.9028} C_DIS
LIN {X 112.4813,Y -38.6961,Z 122,A -22.4586,B 24.9511,C -1.6158,E1 25.1515,E2 468.5045} C_DIS
LIN {X 113.3971,Y -35.924,Z 122,A -21.0573,B 24.9508,C -1.6201,E1 25.1527,E2 467.1012} C_DIS
LIN {X 114.2446,Y -33.1303,Z 122,A -19.5218,B 24.9502,C -1.6309,E1 25.1539,E2 465.5489} C_DIS
LIN {X 115.1723,Y -29.7364,Z 122,A -17.982,B 24.9502,C -1.6288,E1 25.155,E2 464.023} C_DIS
LIN {X 115.8674,Y -26.901,Z 122,A -16.5853,B 24.95,C -1.6328,E1 25.1559,E2 462.6248} C_DIS
LIN {X 116.4927,Y -24.0494,Z 122,A -15.2739,B 24.95,C -1.6328,E1 25.1567,E2 461.3213} C_DIS
LIN {X 117.0478,Y -21.1832,Z 122,A -13.7921,B 24.9495,C -1.641,E1 25.1574,E2 459.8287} C_DIS
LIN {X 117.6639,Y -17.4538,Z 122,A -11.984,B 24.9492,C -1.6463,E1 25.1582,E2 458.0187} C_DIS
LIN {X 118.0568,Y -14.5609,Z 122,A -10.5875,B 24.949,C -1.6504,E1 25.1587,E2 456.6207} C_DIS
LIN {X 118.4128,Y -11.2885,Z 122,A -9.1734,B 24.9492,C -1.6472,E1 25.1591,E2 455.2227} C_DIS
LIN {X 118.6291,Y -8.7506,Z 122,A -7.7944,B 24.9484,C -1.6587,E1 25.1594,E2 453.8247} C_DIS
LIN {X 118.8081,Y -5.8367,Z 122,A -6.398,B 24.9482,C -1.6628,E1 25.1596,E2 452.4269} C_DIS
LIN {X 118.918,Y -2.7871,Z 122,A -4.9057,B 24.9478,C -1.6687,E1 25.1598,E2 450.9296} C_DIS
LIN {X 118.9482,Y 0.6162,Z 122,A -3.2399,B 24.9474,C -1.6754,E1 25.1598,E2 449.258} C_DIS
LIN {X 118.8972,Y 3.518,Z 122,A -1.8864,B 24.9473,C -1.6777,E1 25.1597,E2 447.907} C_DIS
LIN {X 118.7606,Y 6.696,Z 122,A -0.4002,B 24.9471,C -1.6805,E1 25.1595,E2 446.4232} C_DIS
LIN {X 118.5128,Y 10.2057,Z 122,A 1.2829,B 24.9468,C -1.6853,E1 25.1591,E2 444.7385} C_DIS
LIN {X 118.1949,Y 13.382,Z 122,A 2.6923,B 24.9468,C -1.684,E1 25.1587,E2 443.3405} C_DIS
LIN {X 117.8693,Y 16.0086,Z 122,A 4.0764,B 24.9463,C -1.6934,E1 25.1582,E2 441.9424} C_DIS
LIN {X 117.4409,Y 18.8964,Z 122,A 5.4729,B 24.946,C -1.6975,E1 25.1576,E2 440.5446} C_DIS
LIN {X 116.9418,Y 21.7728,Z 122,A 6.8697,B 24.9457,C -1.7015,E1 25.1569,E2 439.1466} C_DIS
LIN {X 116.3722,Y 24.6362,Z 122,A 8.2665,B 24.9455,C -1.7054,E1 25.1561,E2 437.7486} C_DIS
LIN {X 115.7326,Y 27.4847,Z 122,A 9.6634,B 24.9452,C -1.7094,E1 25.1552,E2 436.3505} C_DIS
LIN {X 115.0232,Y 30.3166,Z 122,A 11.0602,B 24.945,C -1.7133,E1 25.1543,E2 434.9525} C_DIS
LIN {X 114.2446,Y 33.1303,Z 122,A 12.4574,B 24.9447,C -1.7172,E1 25.1532,E2 433.5541} C_DIS
LIN {X 113.3971,Y 35.924,Z 122,A 13.8547,B 24.9445,C -1.7211,E1 25.152,E2 432.1557} C_DIS
LIN {X 112.4813,Y 38.6961,Z 122,A 15.3048,B 24.9441,C -1.7275,E1 25.1507,E2 430.6987} C_DIS
LIN {X 111.4978,Y 41.4449,Z 122,A 16.6491,B 24.944,C -1.7286,E1 25.1495,E2 429.3591} C_DIS
LIN {X 110.4471,Y 44.1687,Z 122,A 18.0465,B 24.9438,C -1.7324,E1 25.148,E2 427.9606} C_DIS
LIN {X 109.3299,Y 46.8659,Z 122,A 19.4491,B 24.9435,C -1.7363,E1 25.1465,E2 426.5564} C_DIS
LIN {X 108.1468,Y 49.5349,Z 122,A 20.8415,B 24.9433,C -1.7397,E1 25.1449,E2 425.1636} C_DIS
LIN {X 106.8986,Y 52.174,Z 122,A 22.2393,B 24.943,C -1.7433,E1 25.1432,E2 423.7648} C_DIS
LIN {X 105.586,Y 54.7817,Z 122,A 23.7779,B 24.9424,C -1.7537,E1 25.1412,E2 422.2099} C_DIS
LIN {X 104.2098,Y 57.3564,Z 122,A 25.0351,B 24.9426,C -1.7503,E1 25.1396,E2 420.9672} C_DIS
LIN {X 102.7708,Y 59.8966,Z 122,A 26.4331,B 24.9424,C -1.7538,E1 25.1376,E2 419.5682} C_DIS
LIN {X 101.2699,Y 62.4007,Z 122,A 27.8313,B 24.9421,C -1.7572,E1 25.1356,E2 418.1692} C_DIS
LIN {X 99.708,Y 64.8672,Z 122,A 29.2297,B 24.9419,C -1.7605,E1 25.1335,E2 416.77} C_DIS
LIN {X 98.0861,Y 67.2946,Z 122,A 30.6284,B 24.9417,C -1.7638,E1 25.1313,E2 415.3705} C_DIS
LIN {X 96.1602,Y 70.0158,Z 122,A 32.0461,B 24.942,C -1.7588,E1 25.129,E2 413.9713} C_DIS
LIN {X 94.4308,Y 72.3315,Z 122,A 33.4437,B 24.9418,C -1.7625,E1 25.1267,E2 412.5716} C_DIS
LIN {X 92.8698,Y 74.3279,Z 122,A 34.8247,B 24.9411,C -1.7732,E1 25.1242,E2 411.172} C_DIS
LIN {X 91.0177,Y 76.5847,Z 122,A 36.2237,B 24.9409,C -1.7762,E1 25.1217,E2 409.7724} C_DIS
LIN {X 89.1108,Y 78.7953,Z 122,A 37.623,B 24.9407,C -1.7791,E1 25.1192,E2 408.3724} C_DIS
LIN {X 87.1502,Y 80.9584,Z 122,A 39.0224,B 24.9405,C -1.782,E1 25.1165,E2 406.9725} C_DIS
LIN {X 85.1372,Y 83.0728,Z 122,A 40.4223,B 24.9403,C -1.7848,E1 25.1138,E2 405.572} C_DIS
LIN {X 83.0728,Y 85.1372,Z 122,A 41.8221,B 24.9401,C -1.7875,E1 25.111,E2 404.1717} C_DIS
LIN {X 80.9584,Y 87.1502,Z 122,A 43.222,B 24.9399,C -1.7901,E1 25.1082,E2 402.7713} C_DIS
LIN {X 78.7953,Y 89.1108,Z 122,A 44.7945,B 24.9392,C -1.8009,E1 25.1049,E2 401.1796} C_DIS
LIN {X 76.5847,Y 91.0177,Z 122,A 46.0694,B 24.9394,C -1.7974,E1 25.1022,E2 399.9179} C_DIS
LIN {X 74.3279,Y 92.8698,Z 122,A 47.4231,B 24.9394,C -1.7975,E1 25.0992,E2 398.5689} C_DIS
LIN {X 72.0264,Y 94.6659,Z 122,A 48.9962,B 24.9387,C -1.808,E1 25.0957,E2 396.9769} C_DIS
LIN {X 69.1938,Y 96.753,Z 122,A 50.5124,B 24.9391,C -1.8026,E1 25.0923,E2 395.4789} C_DIS
LIN {X 66.0859,Y 98.9045,Z 122,A 52.3266,B 24.9389,C -1.8053,E1 25.0881,E2 393.6645} C_DIS
LIN {X 63.6387,Y 100.4965,Z 122,A 53.7282,B 24.9388,C -1.8073,E1 25.0849,E2 392.2627} C_DIS
LIN {X 61.1532,Y 102.028,Z 122,A 55.1298,B 24.9386,C -1.8092,E1 25.0815,E2 390.8608} C_DIS
LIN {X 58.6309,Y 103.4981,Z 122,A 56.5317,B 24.9386,C -1.8111,E1 25.0781,E2 389.4588} C_DIS
LIN {X 56.0733,Y 104.9058,Z 122,A 57.9339,B 24.9384,C -1.8128,E1 25.0747,E2 388.0565} C_DIS
LIN {X 53.4819,Y 106.2503,Z 122,A 59.3362,B 24.9383,C -1.8145,E1 25.0712,E2 386.6542} C_DIS
LIN {X 50.8583,Y 107.5308,Z 122,A 60.8706,B 24.9378,C -1.8222,E1 25.0673,E2 385.1056} C_DIS
LIN {X 48.204,Y 108.7465,Z 122,A 62.1415,B 24.9381,C -1.8175,E1 25.0641,E2 383.8489} C_DIS
LIN {X 45.5207,Y 109.8968,Z 122,A 63.5444,B 24.938,C -1.8188,E1 25.0605,E2 382.4461} C_DIS
LIN {X 42.81,Y 110.9808,Z 122,A 64.9476,B 24.938,C -1.8201,E1 25.0568,E2 381.0429} C_DIS
LIN {X 40.0735,Y 111.998,Z 122,A 66.3513,B 24.9378,C -1.8213,E1 25.0531,E2 379.6393} C_DIS
LIN {X 36.8554,Y 113.0957,Z 122,A 68.0178,B 24.9376,C -1.8241,E1 25.0487,E2 377.9695} C_DIS
LIN {X 33.1303,Y 114.2446,Z 122,A 69.8609,B 24.9376,C -1.8238,E1 25.0438,E2 376.1302} C_DIS
LIN {X 30.3166,Y 115.0232,Z 122,A 71.4202,B 24.9371,C -1.8318,E1 25.0395,E2 374.5545} C_DIS
LIN {X 27.4847,Y 115.7326,Z 122,A 72.6694,B 24.9375,C -1.8254,E1 25.0362,E2 373.3222} C_DIS
LIN {X 24.6362,Y 116.3722,Z 122,A 74.0743,B 24.9375,C -1.826,E1 25.0324,E2 371.9177} C_DIS
LIN {X 21.7729,Y 116.9418,Z 122,A 75.4794,B 24.9375,C -1.8266,E1 25.0285,E2 370.513} C_DIS
LIN {X 18.8964,Y 117.4409,Z 122,A 76.8845,B 24.9375,C -1.827,E1 25.0246,E2 369.1083} C_DIS
Enddeposition()
END
